METHOD FB_init : BOOL
VAR_INPUT
	bInitRetains : BOOL; // if TRUE, the retain variables are initialized (warm start / cold start)
	bInCopyCode : BOOL;  // if TRUE, the instance afterwards gets moved into the copy code (online change)
	InitialValue : ETcVnReduceType;
END_VAR
localData := InitialValue;
AddBaseDatatype(enumBaseDatatype);
ClearReference();

AddLocalEnumeration('TCVN_RT_REDUCE_SUM', ETcVnReduceType.TCVN_RT_REDUCE_SUM);
AddLocalEnumeration('TCVN_RT_REDUCE_AVG', ETcVnReduceType.TCVN_RT_REDUCE_AVG);
AddLocalEnumeration('TCVN_RT_REDUCE_MAX', ETcVnReduceType.TCVN_RT_REDUCE_MAX);
AddLocalEnumeration('TCVN_RT_REDUCE_MIN', ETcVnReduceType.TCVN_RT_REDUCE_MIN);
END_METHOD

METHOD PRIVATE AddLocalEnumeration
VAR_INPUT
	Enumeration : T_MAXSTRING;
	Value : ETcVnReduceType;
END_VAR
AddEnumeration(Enumeration, Value);
END_METHOD

METHOD IsEnumeratorValueEqual : BOOL
VAR_INPUT
	Enumerator : I_KeyValueForwardEnumerator;
END_VAR
VAR
	storedValue : ETcVnReduceType;
END_VAR
IF NOT Enumerator.TryGet(storedValue) THEN
	RETURN;
END_IF

IsEnumeratorValueEqual := storedValue = activeData;
END_METHOD

METHOD PUBLIC Clone : I_Datatype
VAR
    pClone : POINTER TO _ETcVnReduceType;
END_VAR
pClone := __NEW(_ETcVnReduceType(InitialValue := Value));
Clone := pClone^;
END_METHOD

PROPERTY PUBLIC Identifier : T_MAXSTRING
GET
Identifier := 'ETcVnReduceType';
END_GET
END_PROPERTY

METHOD PUBLIC MakeReferenceTo
VAR_INPUT
	ReferenceTarget : REFERENCE TO ETcVnReduceType;
END_VAR
activeData REF= ReferenceTarget;
SetBaseDatatypeReference();
END_METHOD

METHOD TryMakeReferenceTo : BOOL
VAR_INPUT
	Target : I_Datatype;
END_VAR
VAR
	pTargetData : POINTER TO ETcVnReduceType;
END_VAR
IF NOT IsEquivalentTo(Target) THEN
	RETURN;
END_IF

pTargetData := Target.Address;
activeData REF= pTargetData^;
SetBaseDatatypeReference();
TryMakeReferenceTo := TRUE;
END_METHOD

PROPERTY PUBLIC Value : ETcVnReduceType
GET
Value := activeData;
END_GET
SET
activeData := Value;
END_SET
END_PROPERTY

END_FUNCTION_BLOCK

// Datatypes/Enums/_ETcVnRotationAngle
{attribute 'linkalways'} 
{attribute 'no_explicit_call' := 'This FB is a CLASS and must be accessed using methods or properties'}
{attribute 'enable_dynamic_creation'}
FUNCTION_BLOCK _ETcVnRotationAngle EXTENDS EnumDatatypeBase
VAR
	localData : ETcVnRotationAngle;
	activeData : REFERENCE TO ETcVnRotationAngle;
	enumBaseDatatype : _DINT(localData);
END_VAR

METHOD PROTECTED SetBaseDatatypeReference
VAR_INPUT
END_VAR
enumBaseDatatype.MakeReferenceTo(activeData);
END_METHOD

PROPERTY PUBLIC Address : PVOID
GET
Address := ADR(activeData);
END_GET
END_PROPERTY

METHOD PUBLIC ClearReference
VAR_INPUT
END_VAR
activeData REF= localData;
SetBaseDatatypeReference();
END_METHOD

PROPERTY PUBLIC Size : UDINT
GET
Size := SIZEOF(activeData);
END_GET
END_PROPERTY

METHOD FB_init : BOOL
VAR_INPUT
	bInitRetains : BOOL; // if TRUE, the retain variables are initialized (warm start / cold start)
	bInCopyCode : BOOL;  // if TRUE, the instance afterwards gets moved into the copy code (online change)
	InitialValue : ETcVnRotationAngle;
END_VAR
localData := InitialValue;
AddBaseDatatype(enumBaseDatatype);
ClearReference();

AddLocalEnumeration('TCVN_RA_90_DEG', ETcVnRotationAngle.TCVN_RA_90_DEG);
AddLocalEnumeration('TCVN_RA_180_DEG', ETcVnRotationAngle.TCVN_RA_180_DEG);
AddLocalEnumeration('TCVN_RA_270_DEG', ETcVnRotationAngle.TCVN_RA_270_DEG);
END_METHOD

METHOD PRIVATE AddLocalEnumeration
VAR_INPUT
	Enumeration : T_MAXSTRING;
	Value : ETcVnRotationAngle;
END_VAR
AddEnumeration(Enumeration, Value);
END_METHOD

METHOD IsEnumeratorValueEqual : BOOL
VAR_INPUT
	Enumerator : I_KeyValueForwardEnumerator;
END_VAR
VAR
	storedValue : ETcVnRotationAngle;
END_VAR
IF NOT Enumerator.TryGet(storedValue) THEN
	RETURN;
END_IF

IsEnumeratorValueEqual := storedValue = activeData;
END_METHOD

METHOD PUBLIC Clone : I_Datatype
VAR
    pClone : POINTER TO _ETcVnRotationAngle;
END_VAR
pClone := __NEW(_ETcVnRotationAngle(InitialValue := Value));
Clone := pClone^;
END_METHOD

PROPERTY PUBLIC Identifier : T_MAXSTRING
GET
Identifier := 'ETcVnRotationAngle';
END_GET
END_PROPERTY

METHOD PUBLIC MakeReferenceTo
VAR_INPUT
	ReferenceTarget : REFERENCE TO ETcVnRotationAngle;
END_VAR
activeData REF= ReferenceTarget;
SetBaseDatatypeReference();
END_METHOD

METHOD TryMakeReferenceTo : BOOL
VAR_INPUT
	Target : I_Datatype;
END_VAR
VAR
	pTargetData : POINTER TO ETcVnRotationAngle;
END_VAR
IF NOT IsEquivalentTo(Target) THEN
	RETURN;
END_IF

pTargetData := Target.Address;
activeData REF= pTargetData^;
SetBaseDatatypeReference();
TryMakeReferenceTo := TRUE;
END_METHOD

PROPERTY PUBLIC Value : ETcVnRotationAngle
GET
Value := activeData;
END_GET
SET
activeData := Value;
END_SET
END_PROPERTY

END_FUNCTION_BLOCK

// Datatypes/Enums/_ETcVnRTrees
{attribute 'linkalways'} 
{attribute 'no_explicit_call' := 'This FB is a CLASS and must be accessed using methods or properties'}
{attribute 'enable_dynamic_creation'}
FUNCTION_BLOCK _ETcVnRTrees EXTENDS EnumDatatypeBase
VAR
	localData : ETcVnRTrees;
	activeData : REFERENCE TO ETcVnRTrees;
	enumBaseDatatype : _UDINT(localData);
END_VAR

METHOD PROTECTED SetBaseDatatypeReference
VAR_INPUT
END_VAR
enumBaseDatatype.MakeReferenceTo(activeData);
END_METHOD

PROPERTY PUBLIC Address : PVOID
GET
Address := ADR(activeData);
END_GET
END_PROPERTY

METHOD PUBLIC ClearReference
VAR_INPUT
END_VAR
activeData REF= localData;
SetBaseDatatypeReference();
END_METHOD

PROPERTY PUBLIC Size : UDINT
GET
Size := SIZEOF(activeData);
END_GET
END_PROPERTY

METHOD FB_init : BOOL
VAR_INPUT
	bInitRetains : BOOL; // if TRUE, the retain variables are initialized (warm start / cold start)
	bInCopyCode : BOOL;  // if TRUE, the instance afterwards gets moved into the copy code (online change)
	InitialValue : ETcVnRTrees;
END_VAR
localData := InitialValue;
AddBaseDatatype(enumBaseDatatype);
ClearReference();

AddLocalEnumeration('TCVN_RT_CLASSIFIER', ETcVnRTrees.TCVN_RT_CLASSIFIER);
AddLocalEnumeration('TCVN_RT_REGRESSOR', ETcVnRTrees.TCVN_RT_REGRESSOR);
END_METHOD

METHOD PRIVATE AddLocalEnumeration
VAR_INPUT
	Enumeration : T_MAXSTRING;
	Value : ETcVnRTrees;
END_VAR
AddEnumeration(Enumeration, Value);
END_METHOD

METHOD IsEnumeratorValueEqual : BOOL
VAR_INPUT
	Enumerator : I_KeyValueForwardEnumerator;
END_VAR
VAR
	storedValue : ETcVnRTrees;
END_VAR
IF NOT Enumerator.TryGet(storedValue) THEN
	RETURN;
END_IF

IsEnumeratorValueEqual := storedValue = activeData;
END_METHOD

METHOD PUBLIC Clone : I_Datatype
VAR
    pClone : POINTER TO _ETcVnRTrees;
END_VAR
pClone := __NEW(_ETcVnRTrees(InitialValue := Value));
Clone := pClone^;
END_METHOD

PROPERTY PUBLIC Identifier : T_MAXSTRING
GET
Identifier := 'ETcVnRTrees';
END_GET
END_PROPERTY

METHOD PUBLIC MakeReferenceTo
VAR_INPUT
	ReferenceTarget : REFERENCE TO ETcVnRTrees;
END_VAR
activeData REF= ReferenceTarget;
SetBaseDatatypeReference();
END_METHOD

METHOD TryMakeReferenceTo : BOOL
VAR_INPUT
	Target : I_Datatype;
END_VAR
VAR
	pTargetData : POINTER TO ETcVnRTrees;
END_VAR
IF NOT IsEquivalentTo(Target) THEN
	RETURN;
END_IF

pTargetData := Target.Address;
activeData REF= pTargetData^;
SetBaseDatatypeReference();
TryMakeReferenceTo := TRUE;
END_METHOD

PROPERTY PUBLIC Value : ETcVnRTrees
GET
Value := activeData;
END_GET
SET
activeData := Value;
END_SET
END_PROPERTY

END_FUNCTION_BLOCK

// Datatypes/Enums/_ETcVnSalientFeaturesMethod
{attribute 'linkalways'}
{attribute 'no_explicit_call' := 'This FB is a CLASS and must be accessed using methods or properties'}
{attribute 'enable_dynamic_creation'}
FUNCTION_BLOCK _ETcVnSalientFeaturesMethod EXTENDS EnumDatatypeBase
VAR
	localData : ETcVnSalientFeaturesMethod;
	activeData : REFERENCE TO ETcVnSalientFeaturesMethod;
	enumBaseDatatype : _UDINT(localData);
END_VAR

METHOD PROTECTED SetBaseDatatypeReference
VAR_INPUT
END_VAR
enumBaseDatatype.MakeReferenceTo(activeData);
END_METHOD

PROPERTY PUBLIC Address : PVOID
GET
Address := ADR(activeData);
END_GET
END_PROPERTY

METHOD PUBLIC ClearReference
VAR_INPUT
END_VAR
activeData REF= localData;
SetBaseDatatypeReference();
END_METHOD

PROPERTY PUBLIC Size : UDINT
GET
Size := SIZEOF(activeData);
END_GET
END_PROPERTY

METHOD FB_init : BOOL
VAR_INPUT
	bInitRetains : BOOL; // if TRUE, the retain variables are initialized (warm start / cold start)
	bInCopyCode : BOOL;  // if TRUE, the instance afterwards gets moved into the copy code (online change)
	InitialValue : ETcVnSalientFeaturesMethod;
END_VAR
localData := InitialValue;
AddBaseDatatype(enumBaseDatatype);
ClearReference();

AddLocalEnumeration('TCVN_SFM_WALSH_CODE', ETcVnSalientFeaturesMethod.TCVN_SFM_WALSH_CODE);
AddLocalEnumeration('TCVN_SFM_SOBEL', ETcVnSalientFeaturesMethod.TCVN_SFM_SOBEL);
END_METHOD

METHOD PRIVATE AddLocalEnumeration
VAR_INPUT
	Enumeration : T_MAXSTRING;
	Value : ETcVnSalientFeaturesMethod;
END_VAR
AddEnumeration(Enumeration, Value);
END_METHOD

METHOD IsEnumeratorValueEqual : BOOL
VAR_INPUT
	Enumerator : I_KeyValueForwardEnumerator;
END_VAR
VAR
	storedValue : ETcVnSalientFeaturesMethod;
END_VAR
IF NOT Enumerator.TryGet(storedValue) THEN
	RETURN;
END_IF

IsEnumeratorValueEqual := storedValue = activeData;
END_METHOD

METHOD PUBLIC Clone : I_Datatype
VAR
    pClone : POINTER TO _ETcVnSalientFeaturesMethod;
END_VAR
pClone := __NEW(_ETcVnSalientFeaturesMethod(InitialValue := Value));
IF pClone = 0 THEN
    RETURN;
END_IF
Clone := pClone^;
END_METHOD

PROPERTY PUBLIC Identifier : T_MAXSTRING
GET
Identifier := 'ETcVnSalientFeaturesMethod';
END_GET
END_PROPERTY

METHOD PUBLIC MakeReferenceTo
VAR_INPUT
	ReferenceTarget : REFERENCE TO ETcVnSalientFeaturesMethod;
END_VAR
activeData REF= ReferenceTarget;
SetBaseDatatypeReference();
END_METHOD

METHOD TryMakeReferenceTo : BOOL
VAR_INPUT
	Target : I_Datatype;
END_VAR
VAR
	pTargetData : POINTER TO ETcVnSalientFeaturesMethod;
END_VAR
IF NOT IsEquivalentTo(Target) THEN
	RETURN;
END_IF

pTargetData := Target.Address;
activeData REF= pTargetData^;
SetBaseDatatypeReference();
TryMakeReferenceTo := TRUE;
END_METHOD

PROPERTY PUBLIC Value : ETcVnSalientFeaturesMethod
GET
Value := activeData;
END_GET
SET
activeData := Value;
END_SET
END_PROPERTY

END_FUNCTION_BLOCK

// Datatypes/Enums/_ETcVnSignedNormalization
{attribute 'linkalways'} 
{attribute 'no_explicit_call' := 'This FB is a CLASS and must be accessed using methods or properties'}
{attribute 'enable_dynamic_creation'}
FUNCTION_BLOCK _ETcVnSignedNormalization EXTENDS EnumDatatypeBase
VAR
	localData : ETcVnSignedNormalization;
	activeData : REFERENCE TO ETcVnSignedNormalization;
	enumBaseDatatype : _INT(localData);
END_VAR

METHOD PROTECTED SetBaseDatatypeReference
VAR_INPUT
END_VAR
enumBaseDatatype.MakeReferenceTo(activeData);
END_METHOD

PROPERTY PUBLIC Address : PVOID
GET
Address := ADR(activeData);
END_GET
END_PROPERTY

METHOD PUBLIC ClearReference
VAR_INPUT
END_VAR
activeData REF= localData;
SetBaseDatatypeReference();
END_METHOD

PROPERTY PUBLIC Size : UDINT
GET
Size := SIZEOF(activeData);
END_GET
END_PROPERTY

METHOD FB_init : BOOL
VAR_INPUT
	bInitRetains : BOOL; // if TRUE, the retain variables are initialized (warm start / cold start)
	bInCopyCode : BOOL;  // if TRUE, the instance afterwards gets moved into the copy code (online change)
	InitialValue : ETcVnSignedNormalization;
END_VAR
localData := InitialValue;
AddBaseDatatype(enumBaseDatatype);
ClearReference();

AddLocalEnumeration('TCVN_SN_FIX_ZERO', ETcVnSignedNormalization.TCVN_SN_FIX_ZERO);
AddLocalEnumeration('TCVN_SN_FULL_SCALE', ETcVnSignedNormalization.TCVN_SN_FULL_SCALE);
END_METHOD

METHOD PRIVATE AddLocalEnumeration
VAR_INPUT
	Enumeration : T_MAXSTRING;
	Value : ETcVnSignedNormalization;
END_VAR
AddEnumeration(Enumeration, Value);
END_METHOD

METHOD IsEnumeratorValueEqual : BOOL
VAR_INPUT
	Enumerator : I_KeyValueForwardEnumerator;
END_VAR
VAR
	storedValue : ETcVnSignedNormalization;
END_VAR
IF NOT Enumerator.TryGet(storedValue) THEN
	RETURN;
END_IF

IsEnumeratorValueEqual := storedValue = activeData;
END_METHOD

METHOD PUBLIC Clone : I_Datatype
VAR
    pClone : POINTER TO _ETcVnSignedNormalization;
END_VAR
pClone := __NEW(_ETcVnSignedNormalization(InitialValue := Value));
Clone := pClone^;
END_METHOD

PROPERTY PUBLIC Identifier : T_MAXSTRING
GET
Identifier := 'ETcVnSignedNormalization';
END_GET
END_PROPERTY

METHOD PUBLIC MakeReferenceTo
VAR_INPUT
	ReferenceTarget : REFERENCE TO ETcVnSignedNormalization;
END_VAR
activeData REF= ReferenceTarget;
SetBaseDatatypeReference();
END_METHOD

METHOD TryMakeReferenceTo : BOOL
VAR_INPUT
	Target : I_Datatype;
END_VAR
VAR
	pTargetData : POINTER TO ETcVnSignedNormalization;
END_VAR
IF NOT IsEquivalentTo(Target) THEN
	RETURN;
END_IF

pTargetData := Target.Address;
activeData REF= pTargetData^;
SetBaseDatatypeReference();
TryMakeReferenceTo := TRUE;
END_METHOD

PROPERTY PUBLIC Value : ETcVnSignedNormalization
GET
Value := activeData;
END_GET
SET
activeData := Value;
END_SET
END_PROPERTY

END_FUNCTION_BLOCK

// Datatypes/Enums/_ETcVnSolvePnPMethod
{attribute 'linkalways'} 
{attribute 'no_explicit_call' := 'This FB is a CLASS and must be accessed using methods or properties'}
{attribute 'enable_dynamic_creation'}
FUNCTION_BLOCK _ETcVnSolvePnPMethod EXTENDS EnumDatatypeBase
VAR
	localData : ETcVnSolvePnPMethod;
	activeData : REFERENCE TO ETcVnSolvePnPMethod;
	enumBaseDatatype : _DINT(localData);
END_VAR

METHOD PROTECTED SetBaseDatatypeReference
VAR_INPUT
END_VAR
enumBaseDatatype.MakeReferenceTo(activeData);
END_METHOD

PROPERTY PUBLIC Address : PVOID
GET
Address := ADR(activeData);
END_GET
END_PROPERTY

METHOD PUBLIC ClearReference
VAR_INPUT
END_VAR
activeData REF= localData;
SetBaseDatatypeReference();
END_METHOD

PROPERTY PUBLIC Size : UDINT
GET
Size := SIZEOF(activeData);
END_GET
END_PROPERTY

METHOD FB_init : BOOL
VAR_INPUT
	bInitRetains : BOOL; // if TRUE, the retain variables are initialized (warm start / cold start)
	bInCopyCode : BOOL;  // if TRUE, the instance afterwards gets moved into the copy code (online change)
	InitialValue : ETcVnSolvePnPMethod;
END_VAR
localData := InitialValue;
AddBaseDatatype(enumBaseDatatype);
ClearReference();

AddLocalEnumeration('TCVN_SPM_ITERATIVE', ETcVnSolvePnPMethod.TCVN_SPM_ITERATIVE);
AddLocalEnumeration('TCVN_SPM_EPNP', ETcVnSolvePnPMethod.TCVN_SPM_EPNP);
AddLocalEnumeration('TCVN_SPM_P3P', ETcVnSolvePnPMethod.TCVN_SPM_P3P);
AddLocalEnumeration('TCVN_SPM_AP3P', ETcVnSolvePnPMethod.TCVN_SPM_AP3P);
AddLocalEnumeration('TCVN_SPM_IPPE', ETcVnSolvePnPMethod.TCVN_SPM_IPPE);
AddLocalEnumeration('TCVN_SPM_IPPE_SQUARE', ETcVnSolvePnPMethod.TCVN_SPM_IPPE_SQUARE);
AddLocalEnumeration('TCVN_SPM_SQPNP', ETcVnSolvePnPMethod.TCVN_SPM_SQPNP);
END_METHOD

METHOD PRIVATE AddLocalEnumeration
VAR_INPUT
	Enumeration : T_MAXSTRING;
	Value : ETcVnSolvePnPMethod;
END_VAR
AddEnumeration(Enumeration, Value);
END_METHOD

METHOD IsEnumeratorValueEqual : BOOL
VAR_INPUT
	Enumerator : I_KeyValueForwardEnumerator;
END_VAR
VAR
	storedValue : ETcVnSolvePnPMethod;
END_VAR
IF NOT Enumerator.TryGet(storedValue) THEN
	RETURN;
END_IF

IsEnumeratorValueEqual := storedValue = activeData;
END_METHOD

METHOD PUBLIC Clone : I_Datatype
VAR
    pClone : POINTER TO _ETcVnSolvePnPMethod;
END_VAR
pClone := __NEW(_ETcVnSolvePnPMethod(InitialValue := Value));
Clone := pClone^;
END_METHOD

PROPERTY PUBLIC Identifier : T_MAXSTRING
GET
Identifier := 'ETcVnSolvePnPMethod';
END_GET
END_PROPERTY

METHOD PUBLIC MakeReferenceTo
VAR_INPUT
	ReferenceTarget : REFERENCE TO ETcVnSolvePnPMethod;
END_VAR
activeData REF= ReferenceTarget;
SetBaseDatatypeReference();
END_METHOD

METHOD TryMakeReferenceTo : BOOL
VAR_INPUT
	Target : I_Datatype;
END_VAR
VAR
	pTargetData : POINTER TO ETcVnSolvePnPMethod;
END_VAR
IF NOT IsEquivalentTo(Target) THEN
	RETURN;
END_IF

pTargetData := Target.Address;
activeData REF= pTargetData^;
SetBaseDatatypeReference();
TryMakeReferenceTo := TRUE;
END_METHOD

PROPERTY PUBLIC Value : ETcVnSolvePnPMethod
GET
Value := activeData;
END_GET
SET
activeData := Value;
END_SET
END_PROPERTY

END_FUNCTION_BLOCK

// Datatypes/Enums/_ETcVnSta
{attribute 'linkalways'} 
{attribute 'no_explicit_call' := 'This FB is a CLASS and must be accessed using methods or properties'}
{attribute 'enable_dynamic_creation'}
FUNCTION_BLOCK _ETcVnSta EXTENDS EnumDatatypeBase
VAR
	localData : ETcVnSta;
	activeData : REFERENCE TO ETcVnSta;
	enumBaseDatatype : _UDINT(localData);
END_VAR

METHOD PROTECTED SetBaseDatatypeReference
VAR_INPUT
END_VAR
enumBaseDatatype.MakeReferenceTo(activeData);
END_METHOD

PROPERTY PUBLIC Address : PVOID
GET
Address := ADR(activeData);
END_GET
END_PROPERTY

METHOD PUBLIC ClearReference
VAR_INPUT
END_VAR
activeData REF= localData;
SetBaseDatatypeReference();
END_METHOD

PROPERTY PUBLIC Size : UDINT
GET
Size := SIZEOF(activeData);
END_GET
END_PROPERTY

METHOD FB_init : BOOL
VAR_INPUT
	bInitRetains : BOOL; // if TRUE, the retain variables are initialized (warm start / cold start)
	bInCopyCode : BOOL;  // if TRUE, the instance afterwards gets moved into the copy code (online change)
	InitialValue : ETcVnSta;
END_VAR
localData := InitialValue;
AddBaseDatatype(enumBaseDatatype);
ClearReference();

AddLocalEnumeration('TCVN_STA_CLASSIFIER', ETcVnSta.TCVN_STA_CLASSIFIER);
AddLocalEnumeration('TCVN_STA_NOVELTY_DETECTOR', ETcVnSta.TCVN_STA_NOVELTY_DETECTOR);
AddLocalEnumeration('TCVN_STA_REGRESSOR', ETcVnSta.TCVN_STA_REGRESSOR);
AddLocalEnumeration('TCVN_STA_CLUSTERER', ETcVnSta.TCVN_STA_CLUSTERER);
END_METHOD

METHOD PRIVATE AddLocalEnumeration
VAR_INPUT
	Enumeration : T_MAXSTRING;
	Value : ETcVnSta;
END_VAR
AddEnumeration(Enumeration, Value);
END_METHOD

METHOD IsEnumeratorValueEqual : BOOL
VAR_INPUT
	Enumerator : I_KeyValueForwardEnumerator;
END_VAR
VAR
	storedValue : ETcVnSta;
END_VAR
IF NOT Enumerator.TryGet(storedValue) THEN
	RETURN;
END_IF

IsEnumeratorValueEqual := storedValue = activeData;
END_METHOD

METHOD PUBLIC Clone : I_Datatype
VAR
    pClone : POINTER TO _ETcVnSta;
END_VAR
pClone := __NEW(_ETcVnSta(InitialValue := Value));
Clone := pClone^;
END_METHOD

PROPERTY PUBLIC Identifier : T_MAXSTRING
GET
Identifier := 'ETcVnSta';
END_GET
END_PROPERTY

METHOD PUBLIC MakeReferenceTo
VAR_INPUT
	ReferenceTarget : REFERENCE TO ETcVnSta;
END_VAR
activeData REF= ReferenceTarget;
SetBaseDatatypeReference();
END_METHOD

METHOD TryMakeReferenceTo : BOOL
VAR_INPUT
	Target : I_Datatype;
END_VAR
VAR
	pTargetData : POINTER TO ETcVnSta;
END_VAR
IF NOT IsEquivalentTo(Target) THEN
	RETURN;
END_IF

pTargetData := Target.Address;
activeData REF= pTargetData^;
SetBaseDatatypeReference();
TryMakeReferenceTo := TRUE;
END_METHOD

PROPERTY PUBLIC Value : ETcVnSta
GET
Value := activeData;
END_GET
SET
activeData := Value;
END_SET
END_PROPERTY

END_FUNCTION_BLOCK

// Datatypes/Enums/_ETcVnStructuringElementShape
{attribute 'linkalways'} 
{attribute 'no_explicit_call' := 'This FB is a CLASS and must be accessed using methods or properties'}
{attribute 'enable_dynamic_creation'}
FUNCTION_BLOCK _ETcVnStructuringElementShape EXTENDS EnumDatatypeBase
VAR
	localData : ETcVnStructuringElementShape;
	activeData : REFERENCE TO ETcVnStructuringElementShape;
	enumBaseDatatype : _DINT(localData);
END_VAR

METHOD PROTECTED SetBaseDatatypeReference
VAR_INPUT
END_VAR
enumBaseDatatype.MakeReferenceTo(activeData);
END_METHOD

PROPERTY PUBLIC Address : PVOID
GET
Address := ADR(activeData);
END_GET
END_PROPERTY

METHOD PUBLIC ClearReference
VAR_INPUT
END_VAR
activeData REF= localData;
SetBaseDatatypeReference();
END_METHOD

PROPERTY PUBLIC Size : UDINT
GET
Size := SIZEOF(activeData);
END_GET
END_PROPERTY

METHOD FB_init : BOOL
VAR_INPUT
	bInitRetains : BOOL; // if TRUE, the retain variables are initialized (warm start / cold start)
	bInCopyCode : BOOL;  // if TRUE, the instance afterwards gets moved into the copy code (online change)
	InitialValue : ETcVnStructuringElementShape;
END_VAR
localData := InitialValue;
AddBaseDatatype(enumBaseDatatype);
ClearReference();

AddLocalEnumeration('TCVN_SES_RECTANGLE', ETcVnStructuringElementShape.TCVN_SES_RECTANGLE);
AddLocalEnumeration('TCVN_SES_CROSS', ETcVnStructuringElementShape.TCVN_SES_CROSS);
AddLocalEnumeration('TCVN_SES_ELLIPSE', ETcVnStructuringElementShape.TCVN_SES_ELLIPSE);
END_METHOD

METHOD PRIVATE AddLocalEnumeration
VAR_INPUT
	Enumeration : T_MAXSTRING;
	Value : ETcVnStructuringElementShape;
END_VAR
AddEnumeration(Enumeration, Value);
END_METHOD

METHOD IsEnumeratorValueEqual : BOOL
VAR_INPUT
	Enumerator : I_KeyValueForwardEnumerator;
END_VAR
VAR
	storedValue : ETcVnStructuringElementShape;
END_VAR
IF NOT Enumerator.TryGet(storedValue) THEN
	RETURN;
END_IF

IsEnumeratorValueEqual := storedValue = activeData;
END_METHOD

METHOD PUBLIC Clone : I_Datatype
VAR
    pClone : POINTER TO _ETcVnStructuringElementShape;
END_VAR
pClone := __NEW(_ETcVnStructuringElementShape(InitialValue := Value));
Clone := pClone^;
END_METHOD

PROPERTY PUBLIC Identifier : T_MAXSTRING
GET
Identifier := 'ETcVnStructuringElementShape';
END_GET
END_PROPERTY

METHOD PUBLIC MakeReferenceTo
VAR_INPUT
	ReferenceTarget : REFERENCE TO ETcVnStructuringElementShape;
END_VAR
activeData REF= ReferenceTarget;
SetBaseDatatypeReference();
END_METHOD

METHOD TryMakeReferenceTo : BOOL
VAR_INPUT
	Target : I_Datatype;
END_VAR
VAR
	pTargetData : POINTER TO ETcVnStructuringElementShape;
END_VAR
IF NOT IsEquivalentTo(Target) THEN
	RETURN;
END_IF

pTargetData := Target.Address;
activeData REF= pTargetData^;
SetBaseDatatypeReference();
TryMakeReferenceTo := TRUE;
END_METHOD

PROPERTY PUBLIC Value : ETcVnStructuringElementShape
GET
Value := activeData;
END_GET
SET
activeData := Value;
END_SET
END_PROPERTY

END_FUNCTION_BLOCK

// Datatypes/Enums/_ETcVnSvm
{attribute 'linkalways'} 
{attribute 'no_explicit_call' := 'This FB is a CLASS and must be accessed using methods or properties'}
{attribute 'enable_dynamic_creation'}
FUNCTION_BLOCK _ETcVnSvm EXTENDS EnumDatatypeBase
VAR
	localData : ETcVnSvm;
	activeData : REFERENCE TO ETcVnSvm;
	enumBaseDatatype : _UDINT(localData);
END_VAR

METHOD PROTECTED SetBaseDatatypeReference
VAR_INPUT
END_VAR
enumBaseDatatype.MakeReferenceTo(activeData);
END_METHOD

PROPERTY PUBLIC Address : PVOID
GET
Address := ADR(activeData);
END_GET
END_PROPERTY

METHOD PUBLIC ClearReference
VAR_INPUT
END_VAR
activeData REF= localData;
SetBaseDatatypeReference();
END_METHOD

PROPERTY PUBLIC Size : UDINT
GET
Size := SIZEOF(activeData);
END_GET
END_PROPERTY

METHOD FB_init : BOOL
VAR_INPUT
	bInitRetains : BOOL; // if TRUE, the retain variables are initialized (warm start / cold start)
	bInCopyCode : BOOL;  // if TRUE, the instance afterwards gets moved into the copy code (online change)
	InitialValue : ETcVnSvm;
END_VAR
localData := InitialValue;
AddBaseDatatype(enumBaseDatatype);
ClearReference();

AddLocalEnumeration('TCVN_SVM_C_CLASSIFIER', ETcVnSvm.TCVN_SVM_C_CLASSIFIER);
AddLocalEnumeration('TCVN_SVM_NU_CLASSIFIER', ETcVnSvm.TCVN_SVM_NU_CLASSIFIER);
AddLocalEnumeration('TCVN_SVM_NOVELTY_DETECTOR', ETcVnSvm.TCVN_SVM_NOVELTY_DETECTOR);
AddLocalEnumeration('TCVN_SVM_EPS_REGRESSOR', ETcVnSvm.TCVN_SVM_EPS_REGRESSOR);
AddLocalEnumeration('TCVN_SVM_NU_REGRESSOR', ETcVnSvm.TCVN_SVM_NU_REGRESSOR);
END_METHOD

METHOD PRIVATE AddLocalEnumeration
VAR_INPUT
	Enumeration : T_MAXSTRING;
	Value : ETcVnSvm;
END_VAR
AddEnumeration(Enumeration, Value);
END_METHOD

METHOD IsEnumeratorValueEqual : BOOL
VAR_INPUT
	Enumerator : I_KeyValueForwardEnumerator;
END_VAR
VAR
	storedValue : ETcVnSvm;
END_VAR
IF NOT Enumerator.TryGet(storedValue) THEN
	RETURN;
END_IF

IsEnumeratorValueEqual := storedValue = activeData;
END_METHOD

METHOD PUBLIC Clone : I_Datatype
VAR
    pClone : POINTER TO _ETcVnSvm;
END_VAR
pClone := __NEW(_ETcVnSvm(InitialValue := Value));
Clone := pClone^;
END_METHOD

PROPERTY PUBLIC Identifier : T_MAXSTRING
GET
Identifier := 'ETcVnSvm';
END_GET
END_PROPERTY

METHOD PUBLIC MakeReferenceTo
VAR_INPUT
	ReferenceTarget : REFERENCE TO ETcVnSvm;
END_VAR
activeData REF= ReferenceTarget;
SetBaseDatatypeReference();
END_METHOD

METHOD TryMakeReferenceTo : BOOL
VAR_INPUT
	Target : I_Datatype;
END_VAR
VAR
	pTargetData : POINTER TO ETcVnSvm;
END_VAR
IF NOT IsEquivalentTo(Target) THEN
	RETURN;
END_IF

pTargetData := Target.Address;
activeData REF= pTargetData^;
SetBaseDatatypeReference();
TryMakeReferenceTo := TRUE;
END_METHOD

PROPERTY PUBLIC Value : ETcVnSvm
GET
Value := activeData;
END_GET
SET
activeData := Value;
END_SET
END_PROPERTY

END_FUNCTION_BLOCK

// Datatypes/Enums/_ETcVnSvmKernelType
{attribute 'linkalways'} 
{attribute 'no_explicit_call' := 'This FB is a CLASS and must be accessed using methods or properties'}
{attribute 'enable_dynamic_creation'}
FUNCTION_BLOCK _ETcVnSvmKernelType EXTENDS EnumDatatypeBase
VAR
	localData : ETcVnSvmKernelType;
	activeData : REFERENCE TO ETcVnSvmKernelType;
	enumBaseDatatype : _DINT(localData);
END_VAR

METHOD PROTECTED SetBaseDatatypeReference
VAR_INPUT
END_VAR
enumBaseDatatype.MakeReferenceTo(activeData);
END_METHOD

PROPERTY PUBLIC Address : PVOID
GET
Address := ADR(activeData);
END_GET
END_PROPERTY

METHOD PUBLIC ClearReference
VAR_INPUT
END_VAR
activeData REF= localData;
SetBaseDatatypeReference();
END_METHOD

PROPERTY PUBLIC Size : UDINT
GET
Size := SIZEOF(activeData);
END_GET
END_PROPERTY

METHOD FB_init : BOOL
VAR_INPUT
	bInitRetains : BOOL; // if TRUE, the retain variables are initialized (warm start / cold start)
	bInCopyCode : BOOL;  // if TRUE, the instance afterwards gets moved into the copy code (online change)
	InitialValue : ETcVnSvmKernelType;
END_VAR
localData := InitialValue;
AddBaseDatatype(enumBaseDatatype);
ClearReference();

AddLocalEnumeration('TCVN_SKT_LINEAR', ETcVnSvmKernelType.TCVN_SKT_LINEAR);
AddLocalEnumeration('TCVN_SKT_POLY', ETcVnSvmKernelType.TCVN_SKT_POLY);
AddLocalEnumeration('TCVN_SKT_RBF', ETcVnSvmKernelType.TCVN_SKT_RBF);
AddLocalEnumeration('TCVN_SKT_SIGMOID', ETcVnSvmKernelType.TCVN_SKT_SIGMOID);
AddLocalEnumeration('TCVN_SKT_CHI2', ETcVnSvmKernelType.TCVN_SKT_CHI2);
AddLocalEnumeration('TCVN_SKT_INTER', ETcVnSvmKernelType.TCVN_SKT_INTER);
END_METHOD

METHOD PRIVATE AddLocalEnumeration
VAR_INPUT
	Enumeration : T_MAXSTRING;
	Value : ETcVnSvmKernelType;
END_VAR
AddEnumeration(Enumeration, Value);
END_METHOD

METHOD IsEnumeratorValueEqual : BOOL
VAR_INPUT
	Enumerator : I_KeyValueForwardEnumerator;
END_VAR
VAR
	storedValue : ETcVnSvmKernelType;
END_VAR
IF NOT Enumerator.TryGet(storedValue) THEN
	RETURN;
END_IF

IsEnumeratorValueEqual := storedValue = activeData;
END_METHOD

METHOD PUBLIC Clone : I_Datatype
VAR
    pClone : POINTER TO _ETcVnSvmKernelType;
END_VAR
pClone := __NEW(_ETcVnSvmKernelType(InitialValue := Value));
Clone := pClone^;
END_METHOD

PROPERTY PUBLIC Identifier : T_MAXSTRING
GET
Identifier := 'ETcVnSvmKernelType';
END_GET
END_PROPERTY

METHOD PUBLIC MakeReferenceTo
VAR_INPUT
	ReferenceTarget : REFERENCE TO ETcVnSvmKernelType;
END_VAR
activeData REF= ReferenceTarget;
SetBaseDatatypeReference();
END_METHOD

METHOD TryMakeReferenceTo : BOOL
VAR_INPUT
	Target : I_Datatype;
END_VAR
VAR
	pTargetData : POINTER TO ETcVnSvmKernelType;
END_VAR
IF NOT IsEquivalentTo(Target) THEN
	RETURN;
END_IF

pTargetData := Target.Address;
activeData REF= pTargetData^;
SetBaseDatatypeReference();
TryMakeReferenceTo := TRUE;
END_METHOD

PROPERTY PUBLIC Value : ETcVnSvmKernelType
GET
Value := activeData;
END_GET
SET
activeData := Value;
END_SET
END_PROPERTY

END_FUNCTION_BLOCK

// Datatypes/Enums/_ETcVnSvmSgdClassifierMarginType
{attribute 'linkalways'} 
{attribute 'no_explicit_call' := 'This FB is a CLASS and must be accessed using methods or properties'}
{attribute 'enable_dynamic_creation'}
FUNCTION_BLOCK _ETcVnSvmSgdClassifierMarginType EXTENDS EnumDatatypeBase
VAR
	localData : ETcVnSvmSgdClassifierMarginType;
	activeData : REFERENCE TO ETcVnSvmSgdClassifierMarginType;
	enumBaseDatatype : _DINT(localData);
END_VAR

METHOD PROTECTED SetBaseDatatypeReference
VAR_INPUT
END_VAR
enumBaseDatatype.MakeReferenceTo(activeData);
END_METHOD

PROPERTY PUBLIC Address : PVOID
GET
Address := ADR(activeData);
END_GET
END_PROPERTY

METHOD PUBLIC ClearReference
VAR_INPUT
END_VAR
activeData REF= localData;
SetBaseDatatypeReference();
END_METHOD

PROPERTY PUBLIC Size : UDINT
GET
Size := SIZEOF(activeData);
END_GET
END_PROPERTY

METHOD FB_init : BOOL
VAR_INPUT
	bInitRetains : BOOL; // if TRUE, the retain variables are initialized (warm start / cold start)
	bInCopyCode : BOOL;  // if TRUE, the instance afterwards gets moved into the copy code (online change)
	InitialValue : ETcVnSvmSgdClassifierMarginType;
END_VAR
localData := InitialValue;
AddBaseDatatype(enumBaseDatatype);
ClearReference();

AddLocalEnumeration('TCVN_SSCMT_SOFT_MARGIN', ETcVnSvmSgdClassifierMarginType.TCVN_SSCMT_SOFT_MARGIN);
AddLocalEnumeration('TCVN_SSCMT_HARD_MARGIN', ETcVnSvmSgdClassifierMarginType.TCVN_SSCMT_HARD_MARGIN);
END_METHOD

METHOD PRIVATE AddLocalEnumeration
VAR_INPUT
	Enumeration : T_MAXSTRING;
	Value : ETcVnSvmSgdClassifierMarginType;
END_VAR
AddEnumeration(Enumeration, Value);
END_METHOD

METHOD IsEnumeratorValueEqual : BOOL
VAR_INPUT
	Enumerator : I_KeyValueForwardEnumerator;
END_VAR
VAR
	storedValue : ETcVnSvmSgdClassifierMarginType;
END_VAR
IF NOT Enumerator.TryGet(storedValue) THEN
	RETURN;
END_IF

IsEnumeratorValueEqual := storedValue = activeData;
END_METHOD

METHOD PUBLIC Clone : I_Datatype
VAR
    pClone : POINTER TO _ETcVnSvmSgdClassifierMarginType;
END_VAR
pClone := __NEW(_ETcVnSvmSgdClassifierMarginType(InitialValue := Value));
Clone := pClone^;
END_METHOD

PROPERTY PUBLIC Identifier : T_MAXSTRING
GET
Identifier := 'ETcVnSvmSgdClassifierMarginType';
END_GET
END_PROPERTY

METHOD PUBLIC MakeReferenceTo
VAR_INPUT
	ReferenceTarget : REFERENCE TO ETcVnSvmSgdClassifierMarginType;
END_VAR
activeData REF= ReferenceTarget;
SetBaseDatatypeReference();
END_METHOD

METHOD TryMakeReferenceTo : BOOL
VAR_INPUT
	Target : I_Datatype;
END_VAR
VAR
	pTargetData : POINTER TO ETcVnSvmSgdClassifierMarginType;
END_VAR
IF NOT IsEquivalentTo(Target) THEN
	RETURN;
END_IF

pTargetData := Target.Address;
activeData REF= pTargetData^;
SetBaseDatatypeReference();
TryMakeReferenceTo := TRUE;
END_METHOD

PROPERTY PUBLIC Value : ETcVnSvmSgdClassifierMarginType
GET
Value := activeData;
END_GET
SET
activeData := Value;
END_SET
END_PROPERTY

END_FUNCTION_BLOCK

// Datatypes/Enums/_ETcVnSvmSgdClassifierType
{attribute 'linkalways'} 
{attribute 'no_explicit_call' := 'This FB is a CLASS and must be accessed using methods or properties'}
{attribute 'enable_dynamic_creation'}
FUNCTION_BLOCK _ETcVnSvmSgdClassifierType EXTENDS EnumDatatypeBase
VAR
	localData : ETcVnSvmSgdClassifierType;
	activeData : REFERENCE TO ETcVnSvmSgdClassifierType;
	enumBaseDatatype : _DINT(localData);
END_VAR

METHOD PROTECTED SetBaseDatatypeReference
VAR_INPUT
END_VAR
enumBaseDatatype.MakeReferenceTo(activeData);
END_METHOD

PROPERTY PUBLIC Address : PVOID
GET
Address := ADR(activeData);
END_GET
END_PROPERTY

METHOD PUBLIC ClearReference
VAR_INPUT
END_VAR
activeData REF= localData;
SetBaseDatatypeReference();
END_METHOD

PROPERTY PUBLIC Size : UDINT
GET
Size := SIZEOF(activeData);
END_GET
END_PROPERTY

METHOD FB_init : BOOL
VAR_INPUT
	bInitRetains : BOOL; // if TRUE, the retain variables are initialized (warm start / cold start)
	bInCopyCode : BOOL;  // if TRUE, the instance afterwards gets moved into the copy code (online change)
	InitialValue : ETcVnSvmSgdClassifierType;
END_VAR
localData := InitialValue;
AddBaseDatatype(enumBaseDatatype);
ClearReference();

AddLocalEnumeration('TCVN_SSCT_SGD', ETcVnSvmSgdClassifierType.TCVN_SSCT_SGD);
AddLocalEnumeration('TCVN_SSCT_ASGD', ETcVnSvmSgdClassifierType.TCVN_SSCT_ASGD);
END_METHOD

METHOD PRIVATE AddLocalEnumeration
VAR_INPUT
	Enumeration : T_MAXSTRING;
	Value : ETcVnSvmSgdClassifierType;
END_VAR
AddEnumeration(Enumeration, Value);
END_METHOD

METHOD IsEnumeratorValueEqual : BOOL
VAR_INPUT
	Enumerator : I_KeyValueForwardEnumerator;
END_VAR
VAR
	storedValue : ETcVnSvmSgdClassifierType;
END_VAR
IF NOT Enumerator.TryGet(storedValue) THEN
	RETURN;
END_IF

IsEnumeratorValueEqual := storedValue = activeData;
END_METHOD

METHOD PUBLIC Clone : I_Datatype
VAR
    pClone : POINTER TO _ETcVnSvmSgdClassifierType;
END_VAR
pClone := __NEW(_ETcVnSvmSgdClassifierType(InitialValue := Value));
Clone := pClone^;
END_METHOD

PROPERTY PUBLIC Identifier : T_MAXSTRING
GET
Identifier := 'ETcVnSvmSgdClassifierType';
END_GET
END_PROPERTY

METHOD PUBLIC MakeReferenceTo
VAR_INPUT
	ReferenceTarget : REFERENCE TO ETcVnSvmSgdClassifierType;
END_VAR
activeData REF= ReferenceTarget;
SetBaseDatatypeReference();
END_METHOD

METHOD TryMakeReferenceTo : BOOL
VAR_INPUT
	Target : I_Datatype;
END_VAR
VAR
	pTargetData : POINTER TO ETcVnSvmSgdClassifierType;
END_VAR
IF NOT IsEquivalentTo(Target) THEN
	RETURN;
END_IF

pTargetData := Target.Address;
activeData REF= pTargetData^;
SetBaseDatatypeReference();
TryMakeReferenceTo := TRUE;
END_METHOD

PROPERTY PUBLIC Value : ETcVnSvmSgdClassifierType
GET
Value := activeData;
END_GET
SET
activeData := Value;
END_SET
END_PROPERTY

END_FUNCTION_BLOCK

// Datatypes/Enums/_ETcVnTemplateMatchMethod
{attribute 'linkalways'} 
{attribute 'no_explicit_call' := 'This FB is a CLASS and must be accessed using methods or properties'}
{attribute 'enable_dynamic_creation'}
FUNCTION_BLOCK _ETcVnTemplateMatchMethod EXTENDS EnumDatatypeBase
VAR
	localData : ETcVnTemplateMatchMethod;
	activeData : REFERENCE TO ETcVnTemplateMatchMethod;
	enumBaseDatatype : _DINT(localData);
END_VAR

METHOD PROTECTED SetBaseDatatypeReference
VAR_INPUT
END_VAR
enumBaseDatatype.MakeReferenceTo(activeData);
END_METHOD

PROPERTY PUBLIC Address : PVOID
GET
Address := ADR(activeData);
END_GET
END_PROPERTY

METHOD PUBLIC ClearReference
VAR_INPUT
END_VAR
activeData REF= localData;
SetBaseDatatypeReference();
END_METHOD

PROPERTY PUBLIC Size : UDINT
GET
Size := SIZEOF(activeData);
END_GET
END_PROPERTY

METHOD FB_init : BOOL
VAR_INPUT
	bInitRetains : BOOL; // if TRUE, the retain variables are initialized (warm start / cold start)
	bInCopyCode : BOOL;  // if TRUE, the instance afterwards gets moved into the copy code (online change)
	InitialValue : ETcVnTemplateMatchMethod;
END_VAR
localData := InitialValue;
AddBaseDatatype(enumBaseDatatype);
ClearReference();

AddLocalEnumeration('TCVN_TMM_SQDIFF', ETcVnTemplateMatchMethod.TCVN_TMM_SQDIFF);
AddLocalEnumeration('TCVN_TMM_SQDIFF_NORMED', ETcVnTemplateMatchMethod.TCVN_TMM_SQDIFF_NORMED);
AddLocalEnumeration('TCVN_TMM_CCORR', ETcVnTemplateMatchMethod.TCVN_TMM_CCORR);
AddLocalEnumeration('TCVN_TMM_CCORR_NORMED', ETcVnTemplateMatchMethod.TCVN_TMM_CCORR_NORMED);
AddLocalEnumeration('TCVN_TMM_CCOEFF', ETcVnTemplateMatchMethod.TCVN_TMM_CCOEFF);
AddLocalEnumeration('TCVN_TMM_CCOEFF_NORMED', ETcVnTemplateMatchMethod.TCVN_TMM_CCOEFF_NORMED);
END_METHOD

METHOD PRIVATE AddLocalEnumeration
VAR_INPUT
	Enumeration : T_MAXSTRING;
	Value : ETcVnTemplateMatchMethod;
END_VAR
AddEnumeration(Enumeration, Value);
END_METHOD

METHOD IsEnumeratorValueEqual : BOOL
VAR_INPUT
	Enumerator : I_KeyValueForwardEnumerator;
END_VAR
VAR
	storedValue : ETcVnTemplateMatchMethod;
END_VAR
IF NOT Enumerator.TryGet(storedValue) THEN
	RETURN;
END_IF

IsEnumeratorValueEqual := storedValue = activeData;
END_METHOD

METHOD PUBLIC Clone : I_Datatype
VAR
    pClone : POINTER TO _ETcVnTemplateMatchMethod;
END_VAR
pClone := __NEW(_ETcVnTemplateMatchMethod(InitialValue := Value));
Clone := pClone^;
END_METHOD

PROPERTY PUBLIC Identifier : T_MAXSTRING
GET
Identifier := 'ETcVnTemplateMatchMethod';
END_GET
END_PROPERTY

METHOD PUBLIC MakeReferenceTo
VAR_INPUT
	ReferenceTarget : REFERENCE TO ETcVnTemplateMatchMethod;
END_VAR
activeData REF= ReferenceTarget;
SetBaseDatatypeReference();
END_METHOD

METHOD TryMakeReferenceTo : BOOL
VAR_INPUT
	Target : I_Datatype;
END_VAR
VAR
	pTargetData : POINTER TO ETcVnTemplateMatchMethod;
END_VAR
IF NOT IsEquivalentTo(Target) THEN
	RETURN;
END_IF

pTargetData := Target.Address;
activeData REF= pTargetData^;
SetBaseDatatypeReference();
TryMakeReferenceTo := TRUE;
END_METHOD

PROPERTY PUBLIC Value : ETcVnTemplateMatchMethod
GET
Value := activeData;
END_GET
SET
activeData := Value;
END_SET
END_PROPERTY

END_FUNCTION_BLOCK

// Datatypes/Enums/_ETcVnThresholdType
{attribute 'linkalways'} 
{attribute 'no_explicit_call' := 'This FB is a CLASS and must be accessed using methods or properties'}
{attribute 'enable_dynamic_creation'}
FUNCTION_BLOCK _ETcVnThresholdType EXTENDS EnumDatatypeBase
VAR
	localData : ETcVnThresholdType;
	activeData : REFERENCE TO ETcVnThresholdType;
	enumBaseDatatype : _DINT(localData);
END_VAR

METHOD PROTECTED SetBaseDatatypeReference
VAR_INPUT
END_VAR
enumBaseDatatype.MakeReferenceTo(activeData);
END_METHOD

PROPERTY PUBLIC Address : PVOID
GET
Address := ADR(activeData);
END_GET
END_PROPERTY

METHOD PUBLIC ClearReference
VAR_INPUT
END_VAR
activeData REF= localData;
SetBaseDatatypeReference();
END_METHOD

PROPERTY PUBLIC Size : UDINT
GET
Size := SIZEOF(activeData);
END_GET
END_PROPERTY

METHOD FB_init : BOOL
VAR_INPUT
	bInitRetains : BOOL; // if TRUE, the retain variables are initialized (warm start / cold start)
	bInCopyCode : BOOL;  // if TRUE, the instance afterwards gets moved into the copy code (online change)
	InitialValue : ETcVnThresholdType;
END_VAR
localData := InitialValue;
AddBaseDatatype(enumBaseDatatype);
ClearReference();

AddLocalEnumeration('TCVN_TT_BINARY', ETcVnThresholdType.TCVN_TT_BINARY);
AddLocalEnumeration('TCVN_TT_BINARY_INV', ETcVnThresholdType.TCVN_TT_BINARY_INV);
AddLocalEnumeration('TCVN_TT_TRUNC', ETcVnThresholdType.TCVN_TT_TRUNC);
AddLocalEnumeration('TCVN_TT_TOZERO', ETcVnThresholdType.TCVN_TT_TOZERO);
AddLocalEnumeration('TCVN_TT_TOZERO_INV', ETcVnThresholdType.TCVN_TT_TOZERO_INV);
AddLocalEnumeration('TCVN_TT_OTSU_BINARY', ETcVnThresholdType.TCVN_TT_OTSU_BINARY);
AddLocalEnumeration('TCVN_TT_OTSU_BINARY_INV', ETcVnThresholdType.TCVN_TT_OTSU_BINARY_INV);
AddLocalEnumeration('TCVN_TT_OTSU_TRUNC', ETcVnThresholdType.TCVN_TT_OTSU_TRUNC);
AddLocalEnumeration('TCVN_TT_OTSU_TOZERO', ETcVnThresholdType.TCVN_TT_OTSU_TOZERO);
AddLocalEnumeration('TCVN_TT_OTSU_TOZERO_INV', ETcVnThresholdType.TCVN_TT_OTSU_TOZERO_INV);
AddLocalEnumeration('TCVN_TT_TRIANGLE_BINARY', ETcVnThresholdType.TCVN_TT_TRIANGLE_BINARY);
AddLocalEnumeration('TCVN_TT_TRIANGLE_BINARY_INV', ETcVnThresholdType.TCVN_TT_TRIANGLE_BINARY_INV);
AddLocalEnumeration('TCVN_TT_TRIANGLE_TRUNC', ETcVnThresholdType.TCVN_TT_TRIANGLE_TRUNC);
AddLocalEnumeration('TCVN_TT_TRIANGLE_TOZERO', ETcVnThresholdType.TCVN_TT_TRIANGLE_TOZERO);
AddLocalEnumeration('TCVN_TT_TRIANGLE_TOZERO_INV', ETcVnThresholdType.TCVN_TT_TRIANGLE_TOZERO_INV);
END_METHOD

METHOD PRIVATE AddLocalEnumeration
VAR_INPUT
	Enumeration : T_MAXSTRING;
	Value : ETcVnThresholdType;
END_VAR
AddEnumeration(Enumeration, Value);
END_METHOD

METHOD IsEnumeratorValueEqual : BOOL
VAR_INPUT
	Enumerator : I_KeyValueForwardEnumerator;
END_VAR
VAR
	storedValue : ETcVnThresholdType;
END_VAR
IF NOT Enumerator.TryGet(storedValue) THEN
	RETURN;
END_IF

IsEnumeratorValueEqual := storedValue = activeData;
END_METHOD

METHOD PUBLIC Clone : I_Datatype
VAR
    pClone : POINTER TO _ETcVnThresholdType;
END_VAR
pClone := __NEW(_ETcVnThresholdType(InitialValue := Value));
Clone := pClone^;
END_METHOD

PROPERTY PUBLIC Identifier : T_MAXSTRING
GET
Identifier := 'ETcVnThresholdType';
END_GET
END_PROPERTY

METHOD PUBLIC MakeReferenceTo
VAR_INPUT
	ReferenceTarget : REFERENCE TO ETcVnThresholdType;
END_VAR
activeData REF= ReferenceTarget;
SetBaseDatatypeReference();
END_METHOD

METHOD TryMakeReferenceTo : BOOL
VAR_INPUT
	Target : I_Datatype;
END_VAR
VAR
	pTargetData : POINTER TO ETcVnThresholdType;
END_VAR
IF NOT IsEquivalentTo(Target) THEN
	RETURN;
END_IF

pTargetData := Target.Address;
activeData REF= pTargetData^;
SetBaseDatatypeReference();
TryMakeReferenceTo := TRUE;
END_METHOD

PROPERTY PUBLIC Value : ETcVnThresholdType
GET
Value := activeData;
END_GET
SET
activeData := Value;
END_SET
END_PROPERTY

END_FUNCTION_BLOCK

// Datatypes/Enums/_ETcVnTimestamp
{attribute 'linkalways'} 
{attribute 'no_explicit_call' := 'This FB is a CLASS and must be accessed using methods or properties'}
{attribute 'enable_dynamic_creation'}
FUNCTION_BLOCK _ETcVnTimestamp EXTENDS EnumDatatypeBase
VAR
	localData : ETcVnTimestamp;
	activeData : REFERENCE TO ETcVnTimestamp;
	enumBaseDatatype : _ULINT(localData);
END_VAR

METHOD PROTECTED SetBaseDatatypeReference
VAR_INPUT
END_VAR
enumBaseDatatype.MakeReferenceTo(activeData);
END_METHOD

PROPERTY PUBLIC Address : PVOID
GET
Address := ADR(activeData);
END_GET
END_PROPERTY

METHOD PUBLIC ClearReference
VAR_INPUT
END_VAR
activeData REF= localData;
SetBaseDatatypeReference();
END_METHOD

PROPERTY PUBLIC Size : UDINT
GET
Size := SIZEOF(activeData);
END_GET
END_PROPERTY

METHOD FB_init : BOOL
VAR_INPUT
	bInitRetains : BOOL; // if TRUE, the retain variables are initialized (warm start / cold start)
	bInCopyCode : BOOL;  // if TRUE, the instance afterwards gets moved into the copy code (online change)
	InitialValue : ETcVnTimestamp;
END_VAR
localData := InitialValue;
AddBaseDatatype(enumBaseDatatype);
ClearReference();

AddLocalEnumeration('TCVN_TS_IMAGE_COMPLETED', ETcVnTimestamp.TCVN_TS_IMAGE_COMPLETED);
AddLocalEnumeration('TCVN_TS_RECEPTION_STARTED', ETcVnTimestamp.TCVN_TS_RECEPTION_STARTED);
AddLocalEnumeration('TCVN_TS_RECEPTION_FINISHED', ETcVnTimestamp.TCVN_TS_RECEPTION_FINISHED);
AddLocalEnumeration('TCVN_TS_GETCURRENTIMAGE', ETcVnTimestamp.TCVN_TS_GETCURRENTIMAGE);
AddLocalEnumeration('TCVN_TS_CAMERA', ETcVnTimestamp.TCVN_TS_CAMERA);
AddLocalEnumeration('TCVN_TS_CUSTOM', ETcVnTimestamp.TCVN_TS_CUSTOM);
AddLocalEnumeration('TCVN_TS_LAST_CHANGE', ETcVnTimestamp.TCVN_TS_LAST_CHANGE);
END_METHOD

METHOD PRIVATE AddLocalEnumeration
VAR_INPUT
	Enumeration : T_MAXSTRING;
	Value : ETcVnTimestamp;
END_VAR
AddEnumeration(Enumeration, Value);
END_METHOD

METHOD IsEnumeratorValueEqual : BOOL
VAR_INPUT
	Enumerator : I_KeyValueForwardEnumerator;
END_VAR
VAR
	storedValue : ETcVnTimestamp;
END_VAR
IF NOT Enumerator.TryGet(storedValue) THEN
	RETURN;
END_IF

IsEnumeratorValueEqual := storedValue = activeData;
END_METHOD

METHOD PUBLIC Clone : I_Datatype
VAR
    pClone : POINTER TO _ETcVnTimestamp;
END_VAR
pClone := __NEW(_ETcVnTimestamp(InitialValue := Value));
Clone := pClone^;
END_METHOD

PROPERTY PUBLIC Identifier : T_MAXSTRING
GET
Identifier := 'ETcVnTimestamp';
END_GET
END_PROPERTY

METHOD PUBLIC MakeReferenceTo
VAR_INPUT
	ReferenceTarget : REFERENCE TO ETcVnTimestamp;
END_VAR
activeData REF= ReferenceTarget;
SetBaseDatatypeReference();
END_METHOD

METHOD TryMakeReferenceTo : BOOL
VAR_INPUT
	Target : I_Datatype;
END_VAR
VAR
	pTargetData : POINTER TO ETcVnTimestamp;
END_VAR
IF NOT IsEquivalentTo(Target) THEN
	RETURN;
END_IF

pTargetData := Target.Address;
activeData REF= pTargetData^;
SetBaseDatatypeReference();
TryMakeReferenceTo := TRUE;
END_METHOD

PROPERTY PUBLIC Value : ETcVnTimestamp
GET
Value := activeData;
END_GET
SET
activeData := Value;
END_SET
END_PROPERTY

END_FUNCTION_BLOCK

// Datatypes/Enums/_ETcVnVectorCompareMethod
{attribute 'linkalways'} 
{attribute 'no_explicit_call' := 'This FB is a CLASS and must be accessed using methods or properties'}
{attribute 'enable_dynamic_creation'}
FUNCTION_BLOCK _ETcVnVectorCompareMethod EXTENDS EnumDatatypeBase
VAR
	localData : ETcVnVectorCompareMethod;
	activeData : REFERENCE TO ETcVnVectorCompareMethod;
	enumBaseDatatype : _DINT(localData);
END_VAR

METHOD PROTECTED SetBaseDatatypeReference
VAR_INPUT
END_VAR
enumBaseDatatype.MakeReferenceTo(activeData);
END_METHOD

PROPERTY PUBLIC Address : PVOID
GET
Address := ADR(activeData);
END_GET
END_PROPERTY

METHOD PUBLIC ClearReference
VAR_INPUT
END_VAR
activeData REF= localData;
SetBaseDatatypeReference();
END_METHOD

PROPERTY PUBLIC Size : UDINT
GET
Size := SIZEOF(activeData);
END_GET
END_PROPERTY

METHOD FB_init : BOOL
VAR_INPUT
	bInitRetains : BOOL; // if TRUE, the retain variables are initialized (warm start / cold start)
	bInCopyCode : BOOL;  // if TRUE, the instance afterwards gets moved into the copy code (online change)
	InitialValue : ETcVnVectorCompareMethod;
END_VAR
localData := InitialValue;
AddBaseDatatype(enumBaseDatatype);
ClearReference();

AddLocalEnumeration('TCVN_VCM_EUCLIDEAN', ETcVnVectorCompareMethod.TCVN_VCM_EUCLIDEAN);
AddLocalEnumeration('TCVN_VCM_ELEMENTWISE', ETcVnVectorCompareMethod.TCVN_VCM_ELEMENTWISE);
END_METHOD

METHOD PRIVATE AddLocalEnumeration
VAR_INPUT
	Enumeration : T_MAXSTRING;
	Value : ETcVnVectorCompareMethod;
END_VAR
AddEnumeration(Enumeration, Value);
END_METHOD

METHOD IsEnumeratorValueEqual : BOOL
VAR_INPUT
	Enumerator : I_KeyValueForwardEnumerator;
END_VAR
VAR
	storedValue : ETcVnVectorCompareMethod;
END_VAR
IF NOT Enumerator.TryGet(storedValue) THEN
	RETURN;
END_IF

IsEnumeratorValueEqual := storedValue = activeData;
END_METHOD

METHOD PUBLIC Clone : I_Datatype
VAR
    pClone : POINTER TO _ETcVnVectorCompareMethod;
END_VAR
pClone := __NEW(_ETcVnVectorCompareMethod(InitialValue := Value));
Clone := pClone^;
END_METHOD

PROPERTY PUBLIC Identifier : T_MAXSTRING
GET
Identifier := 'ETcVnVectorCompareMethod';
END_GET
END_PROPERTY

METHOD PUBLIC MakeReferenceTo
VAR_INPUT
	ReferenceTarget : REFERENCE TO ETcVnVectorCompareMethod;
END_VAR
activeData REF= ReferenceTarget;
SetBaseDatatypeReference();
END_METHOD

METHOD TryMakeReferenceTo : BOOL
VAR_INPUT
	Target : I_Datatype;
END_VAR
VAR
	pTargetData : POINTER TO ETcVnVectorCompareMethod;
END_VAR
IF NOT IsEquivalentTo(Target) THEN
	RETURN;
END_IF

pTargetData := Target.Address;
activeData REF= pTargetData^;
SetBaseDatatypeReference();
TryMakeReferenceTo := TRUE;
END_METHOD

PROPERTY PUBLIC Value : ETcVnVectorCompareMethod
GET
Value := activeData;
END_GET
SET
activeData := Value;
END_SET
END_PROPERTY

END_FUNCTION_BLOCK

// Datatypes/Enums/_ETcVnWorldCoordinateSystem
{attribute 'linkalways'} 
{attribute 'no_explicit_call' := 'This FB is a CLASS and must be accessed using methods or properties'}
{attribute 'enable_dynamic_creation'}
FUNCTION_BLOCK _ETcVnWorldCoordinateSystem EXTENDS EnumDatatypeBase
VAR
	localData : ETcVnWorldCoordinateSystem;
	activeData : REFERENCE TO ETcVnWorldCoordinateSystem;
	enumBaseDatatype : _DINT(localData);
END_VAR

METHOD PROTECTED SetBaseDatatypeReference
VAR_INPUT
END_VAR
enumBaseDatatype.MakeReferenceTo(activeData);
END_METHOD

PROPERTY PUBLIC Address : PVOID
GET
Address := ADR(activeData);
END_GET
END_PROPERTY

METHOD PUBLIC ClearReference
VAR_INPUT
END_VAR
activeData REF= localData;
SetBaseDatatypeReference();
END_METHOD

PROPERTY PUBLIC Size : UDINT
GET
Size := SIZEOF(activeData);
END_GET
END_PROPERTY

METHOD FB_init : BOOL
VAR_INPUT
	bInitRetains : BOOL; // if TRUE, the retain variables are initialized (warm start / cold start)
	bInCopyCode : BOOL;  // if TRUE, the instance afterwards gets moved into the copy code (online change)
	InitialValue : ETcVnWorldCoordinateSystem;
END_VAR
localData := InitialValue;
AddBaseDatatype(enumBaseDatatype);
ClearReference();

AddLocalEnumeration('TCVN_WCS_X_RIGHT_Y_DOWN' , ETcVnWorldCoordinateSystem.TCVN_WCS_X_RIGHT_Y_DOWN);
AddLocalEnumeration('TCVN_WCS_X_DOWN_Y_RIGHT', ETcVnWorldCoordinateSystem.TCVN_WCS_X_DOWN_Y_RIGHT);
AddLocalEnumeration('TCVN_WCS_X_LEFT_Y_DOWN', ETcVnWorldCoordinateSystem.TCVN_WCS_X_LEFT_Y_DOWN);
AddLocalEnumeration('TCVN_WCS_X_UP_Y_RIGHT', ETcVnWorldCoordinateSystem.TCVN_WCS_X_UP_Y_RIGHT);
AddLocalEnumeration('TCVN_WCS_X_RIGHT_Y_UP', ETcVnWorldCoordinateSystem.TCVN_WCS_X_RIGHT_Y_UP);
AddLocalEnumeration('TCVN_WCS_X_DOWN_Y_LEFT', ETcVnWorldCoordinateSystem.TCVN_WCS_X_DOWN_Y_LEFT);
AddLocalEnumeration('TCVN_WCS_X_LEFT_Y_UP', ETcVnWorldCoordinateSystem.TCVN_WCS_X_LEFT_Y_UP);
AddLocalEnumeration('TCVN_WCS_X_UP_Y_LEFT', ETcVnWorldCoordinateSystem.TCVN_WCS_X_UP_Y_LEFT);
END_METHOD

METHOD PRIVATE AddLocalEnumeration
VAR_INPUT
	Enumeration : T_MAXSTRING;
	Value : ETcVnWorldCoordinateSystem;
END_VAR
AddEnumeration(Enumeration, Value);
END_METHOD

METHOD IsEnumeratorValueEqual : BOOL
VAR_INPUT
	Enumerator : I_KeyValueForwardEnumerator;
END_VAR
VAR
	storedValue : ETcVnWorldCoordinateSystem;
END_VAR
IF NOT Enumerator.TryGet(storedValue) THEN
	RETURN;
END_IF

IsEnumeratorValueEqual := storedValue = activeData;
END_METHOD

METHOD PUBLIC Clone : I_Datatype
VAR
    pClone : POINTER TO _ETcVnWorldCoordinateSystem;
END_VAR
pClone := __NEW(_ETcVnWorldCoordinateSystem(InitialValue := Value));
Clone := pClone^;
END_METHOD

PROPERTY PUBLIC Identifier : T_MAXSTRING
GET
Identifier := 'ETcVnWorldCoordinateSystem';
END_GET
END_PROPERTY

METHOD PUBLIC MakeReferenceTo
VAR_INPUT
	ReferenceTarget : REFERENCE TO ETcVnWorldCoordinateSystem;
END_VAR
activeData REF= ReferenceTarget;
SetBaseDatatypeReference();
END_METHOD

METHOD TryMakeReferenceTo : BOOL
VAR_INPUT
	Target : I_Datatype;
END_VAR
VAR
	pTargetData : POINTER TO ETcVnWorldCoordinateSystem;
END_VAR
IF NOT IsEquivalentTo(Target) THEN
	RETURN;
END_IF

pTargetData := Target.Address;
activeData REF= pTargetData^;
SetBaseDatatypeReference();
TryMakeReferenceTo := TRUE;
END_METHOD

PROPERTY PUBLIC Value : ETcVnWorldCoordinateSystem
GET
Value := activeData;
END_GET
SET
activeData := Value;
END_SET
END_PROPERTY

END_FUNCTION_BLOCK

// Datatypes/Enums/_ETcWatchdogAccumulationType
{attribute 'linkalways'} 
{attribute 'no_explicit_call' := 'This FB is a CLASS and must be accessed using methods or properties'}
{attribute 'enable_dynamic_creation'}
FUNCTION_BLOCK _ETcWatchdogAccumulationType EXTENDS EnumDatatypeBase
VAR
	localData : ETcWatchdogAccumulationType;
	activeData : REFERENCE TO ETcWatchdogAccumulationType;
	enumBaseDatatype : _UINT(localData);
END_VAR

METHOD PROTECTED SetBaseDatatypeReference
VAR_INPUT
END_VAR
enumBaseDatatype.MakeReferenceTo(activeData);
END_METHOD

PROPERTY PUBLIC Address : PVOID
GET
Address := ADR(activeData);
END_GET
END_PROPERTY

METHOD PUBLIC ClearReference
VAR_INPUT
END_VAR
activeData REF= localData;
SetBaseDatatypeReference();
END_METHOD

PROPERTY PUBLIC Size : UDINT
GET
Size := SIZEOF(activeData);
END_GET
END_PROPERTY

METHOD FB_init : BOOL
VAR_INPUT
	bInitRetains : BOOL; // if TRUE, the retain variables are initialized (warm start / cold start)
	bInCopyCode : BOOL;  // if TRUE, the instance afterwards gets moved into the copy code (online change)
	InitialValue : ETcWatchdogAccumulationType;
END_VAR
localData := InitialValue;
AddBaseDatatype(enumBaseDatatype);
ClearReference();

AddLocalEnumeration('WD_ACC_TYPE_MEAN', ETcWatchdogAccumulationType.WD_ACC_TYPE_MEAN);
AddLocalEnumeration('WD_ACC_TYPE_PRODUCT', ETcWatchdogAccumulationType.WD_ACC_TYPE_PRODUCT);
END_METHOD

METHOD PRIVATE AddLocalEnumeration
VAR_INPUT
	Enumeration : T_MAXSTRING;
	Value : ETcWatchdogAccumulationType;
END_VAR
AddEnumeration(Enumeration, Value);
END_METHOD

METHOD IsEnumeratorValueEqual : BOOL
VAR_INPUT
	Enumerator : I_KeyValueForwardEnumerator;
END_VAR
VAR
	storedValue : ETcWatchdogAccumulationType;
END_VAR
IF NOT Enumerator.TryGet(storedValue) THEN
	RETURN;
END_IF

IsEnumeratorValueEqual := storedValue = activeData;
END_METHOD

METHOD PUBLIC Clone : I_Datatype
VAR
    pClone : POINTER TO _ETcWatchdogAccumulationType;
END_VAR
pClone := __NEW(_ETcWatchdogAccumulationType(InitialValue := Value));
Clone := pClone^;
END_METHOD

PROPERTY PUBLIC Identifier : T_MAXSTRING
GET
Identifier := 'ETcWatchdogAccumulationType';
END_GET
END_PROPERTY

METHOD PUBLIC MakeReferenceTo
VAR_INPUT
	ReferenceTarget : REFERENCE TO ETcWatchdogAccumulationType;
END_VAR
activeData REF= ReferenceTarget;
SetBaseDatatypeReference();
END_METHOD

METHOD TryMakeReferenceTo : BOOL
VAR_INPUT
	Target : I_Datatype;
END_VAR
VAR
	pTargetData : POINTER TO ETcWatchdogAccumulationType;
END_VAR
IF NOT IsEquivalentTo(Target) THEN
	RETURN;
END_IF

pTargetData := Target.Address;
activeData REF= pTargetData^;
SetBaseDatatypeReference();
TryMakeReferenceTo := TRUE;
END_METHOD

PROPERTY PUBLIC Value : ETcWatchdogAccumulationType
GET
Value := activeData;
END_GET
SET
activeData := Value;
END_SET
END_PROPERTY

END_FUNCTION_BLOCK

// Datatypes/Enums/_GEV_CAMERA_STATE
{attribute 'linkalways'} 
{attribute 'no_explicit_call' := 'This FB is a CLASS and must be accessed using methods or properties'}
{attribute 'enable_dynamic_creation'}
FUNCTION_BLOCK _GEV_CAMERA_STATE EXTENDS EnumDatatypeBase
VAR
	localData : GEV_CAMERA_STATE;
	activeData : REFERENCE TO GEV_CAMERA_STATE;
	enumBaseDatatype : _BYTE(localData);
END_VAR

METHOD PROTECTED SetBaseDatatypeReference
VAR_INPUT
END_VAR
enumBaseDatatype.MakeReferenceTo(activeData);
END_METHOD

PROPERTY PUBLIC Address : PVOID
GET
Address := ADR(activeData);
END_GET
END_PROPERTY

METHOD PUBLIC ClearReference
VAR_INPUT
END_VAR
activeData REF= localData;
SetBaseDatatypeReference();
END_METHOD

PROPERTY PUBLIC Size : UDINT
GET
Size := SIZEOF(activeData);
END_GET
END_PROPERTY

METHOD FB_init : BOOL
VAR_INPUT
	bInitRetains : BOOL; // if TRUE, the retain variables are initialized (warm start / cold start)
	bInCopyCode : BOOL;  // if TRUE, the instance afterwards gets moved into the copy code (online change)
	InitialValue : GEV_CAMERA_STATE;
END_VAR
localData := InitialValue;
AddBaseDatatype(enumBaseDatatype);
ClearReference();

AddLocalEnumeration('GEV_CAMERA_IDLE', GEV_CAMERA_STATE.GEV_CAMERA_IDLE);
AddLocalEnumeration('GEV_CONTROL_CHANNEL_OPEN_MASK', GEV_CAMERA_STATE.GEV_CONTROL_CHANNEL_OPEN_MASK);
AddLocalEnumeration('GEV_STREAM_CHANNELS_OPEN_MASK', GEV_CAMERA_STATE.GEV_STREAM_CHANNELS_OPEN_MASK);
AddLocalEnumeration('GEV_CONTROL_CHANNEL_OPEN', GEV_CAMERA_STATE.GEV_CONTROL_CHANNEL_OPEN);
AddLocalEnumeration('GEV_STREAM_CHANNELS_OPEN', GEV_CAMERA_STATE.GEV_STREAM_CHANNELS_OPEN);
END_METHOD

METHOD PRIVATE AddLocalEnumeration
VAR_INPUT
	Enumeration : T_MAXSTRING;
	Value : GEV_CAMERA_STATE;
END_VAR
AddEnumeration(Enumeration, Value);
END_METHOD

METHOD IsEnumeratorValueEqual : BOOL
VAR_INPUT
	Enumerator : I_KeyValueForwardEnumerator;
END_VAR
VAR
	storedValue : GEV_CAMERA_STATE;
END_VAR
IF NOT Enumerator.TryGet(storedValue) THEN
	RETURN;
END_IF

IsEnumeratorValueEqual := storedValue = activeData;
END_METHOD

METHOD PUBLIC Clone : I_Datatype
VAR
    pClone : POINTER TO _GEV_CAMERA_STATE;
END_VAR
pClone := __NEW(_GEV_CAMERA_STATE(InitialValue := Value));
Clone := pClone^;
END_METHOD

PROPERTY PUBLIC Identifier : T_MAXSTRING
GET
Identifier := 'GEV_CAMERA_STATE';
END_GET
END_PROPERTY

METHOD PUBLIC MakeReferenceTo
VAR_INPUT
	ReferenceTarget : REFERENCE TO GEV_CAMERA_STATE;
END_VAR
activeData REF= ReferenceTarget;
SetBaseDatatypeReference();
END_METHOD

METHOD TryMakeReferenceTo : BOOL
VAR_INPUT
	Target : I_Datatype;
END_VAR
VAR
	pTargetData : POINTER TO GEV_CAMERA_STATE;
END_VAR
IF NOT IsEquivalentTo(Target) THEN
	RETURN;
END_IF

pTargetData := Target.Address;
activeData REF= pTargetData^;
SetBaseDatatypeReference();
TryMakeReferenceTo := TRUE;
END_METHOD

PROPERTY PUBLIC Value : GEV_CAMERA_STATE
GET
Value := activeData;
END_GET
SET
activeData := Value;
END_SET
END_PROPERTY

END_FUNCTION_BLOCK

// Datatypes/Interfaces/Containers/ITcVnContainer/_ITcVnContainer
{attribute 'linkalways'} 
{attribute 'no_explicit_call' := 'This FB is a CLASS and must be accessed using methods or properties'}
{attribute 'enable_dynamic_creation'}
FUNCTION_BLOCK _ITcVnContainer EXTENDS InterfaceDatatypeBase IMPLEMENTS I_InterfaceDatatype_ITcVnContainer
VAR
	localData : ITcVnContainer;
	activeData : REFERENCE TO ITcVnContainer REF= localData;
END_VAR

PROPERTY PUBLIC Address : PVOID
GET
Address := ADR(activeData);
END_GET
END_PROPERTY

METHOD PUBLIC ClearReference
VAR_INPUT
END_VAR
activeData REF= localData;
END_METHOD

PROPERTY PUBLIC Size : UDINT
GET
Size := SIZEOF(activeData);
END_GET
END_PROPERTY

METHOD FB_exit : BOOL
VAR_INPUT
	bInCopyCode : BOOL; // if TRUE, the exit method is called for exiting an instance that is copied afterwards (online change).
END_VAR
IF bInCopyCode THEN
	RETURN;
END_IF

TryTcReleaseLocal();
END_METHOD

METHOD PRIVATE Serialize_ContainerType_String_SINT
VAR_INPUT
	Serializer : I_Serializer;
	TargetContainer : ITcVnContainer;
END_VAR
VAR
	hr : HRESULT;
	_value : _STRING('');
END_VAR
hr := F_VN_ExportContainer_String(TargetContainer, _value.Value, SIZEOF(_value.Value), S_OK);
Serializer.StartArray();

IF SUCCEEDED(hr) THEN
	Serializer.AddObject(_value);
ELSE
	Serializer.AddNull();
END_IF

Serializer.EndArray();
END_METHOD

METHOD PRIVATE Serialize_ContainerType_Vector_DINT
VAR_INPUT
	Serializer : I_Serializer;
	TargetContainer : ITcVnContainer;
END_VAR
VAR
	hr : HRESULT;
	_value : _DINT(0);
	elementCount : ULINT;
	i : ULINT;
END_VAR
TargetContainer.GetElementNum(elementCount);
Serializer.StartArray();

IF elementCount > 0 THEN
	FOR i := 0 TO elementCount - 1 DO 
		
		hr := F_VN_GetAt_DINT(TargetContainer, _value.Value, i, S_OK);
		
		IF SUCCEEDED(hr) THEN
			Serializer.AddObject(_value);
		ELSE
			Serializer.AddNull();
		END_IF
		
	END_FOR
END_IF

Serializer.EndArray();
END_METHOD

METHOD PRIVATE Serialize_ContainerType_Vector_INT
VAR_INPUT
	Serializer : I_Serializer;
	TargetContainer : ITcVnContainer;
END_VAR
VAR
	hr : HRESULT;
	_value : _INT(0);
	elementCount : ULINT;
	i : ULINT;
END_VAR
TargetContainer.GetElementNum(elementCount);
Serializer.StartArray();

IF elementCount > 0 THEN
	FOR i := 0 TO elementCount - 1 DO 
		
		hr := F_VN_GetAt_INT(TargetContainer, _value.Value, i, S_OK);
		
		IF SUCCEEDED(hr) THEN
			Serializer.AddObject(_value);
		ELSE
			Serializer.AddNull();
		END_IF
		
	END_FOR
END_IF

Serializer.EndArray();
END_METHOD

METHOD PRIVATE Serialize_ContainerType_Vector_ITcVnImage
VAR_INPUT
	Serializer : I_Serializer;
	TargetContainer : ITcVnContainer;
END_VAR
VAR
	hr : HRESULT;
	_value : _ITcVnImage;
	elementCount : ULINT;
	i : ULINT;
END_VAR
TargetContainer.GetElementNum(elementCount);
Serializer.StartArray();

IF elementCount > 0 THEN
	FOR i := 0 TO elementCount - 1 DO 
		
		hr := F_VN_GetAt_ITcVnImage(TargetContainer, _value.Value, i, S_OK);
		
		IF SUCCEEDED(hr) THEN
			Serializer.AddObject(_value);
		ELSE
			Serializer.AddNull();
		END_IF
	
	END_FOR
END_IF

IF _value.Value <> 0 THEN
	_value.Value.TcRelease();
END_IF

Serializer.EndArray();
END_METHOD

METHOD PRIVATE Serialize_ContainerType_Vector_LREAL
VAR_INPUT
	Serializer : I_Serializer;
	TargetContainer : ITcVnContainer;
END_VAR
VAR
	hr : HRESULT;
	_value : _LREAL(0);
	elementCount : ULINT;
	i : ULINT;
END_VAR
TargetContainer.GetElementNum(elementCount);
Serializer.StartArray();

IF elementCount > 0 THEN
	FOR i := 0 TO elementCount - 1 DO 
		
		hr := F_VN_GetAt_LREAL(TargetContainer, _value.Value, i, S_OK);
		
		IF SUCCEEDED(hr) THEN
			Serializer.AddObject(_value);
		ELSE
			Serializer.AddNull();
		END_IF
		
	END_FOR
END_IF

Serializer.EndArray();
END_METHOD

METHOD PRIVATE Serialize_ContainerType_Vector_REAL
VAR_INPUT
	Serializer : I_Serializer;
	TargetContainer : ITcVnContainer;
END_VAR
VAR
	hr : HRESULT;
	_value : _REAL(0);
	elementCount : ULINT;
	i : ULINT;
END_VAR
TargetContainer.GetElementNum(elementCount);
Serializer.StartArray();

IF elementCount > 0 THEN
	FOR i := 0 TO elementCount - 1 DO 
		
		hr := F_VN_GetAt_REAL(TargetContainer, _value.Value, i, S_OK);
		
		IF SUCCEEDED(hr) THEN
			Serializer.AddObject(_value);
		ELSE
			Serializer.AddNull();
		END_IF
		
	END_FOR
END_IF

Serializer.EndArray();
END_METHOD

METHOD PRIVATE Serialize_ContainerType_Vector_SINT
VAR_INPUT
	Serializer : I_Serializer;
	TargetContainer : ITcVnContainer;
END_VAR
VAR
	hr : HRESULT;
	_value : _SINT(0);
	elementCount : ULINT;
	i : ULINT;
END_VAR
TargetContainer.GetElementNum(elementCount);
Serializer.StartArray();

IF elementCount > 0 THEN
	FOR i := 0 TO elementCount - 1 DO 
		
		hr := F_VN_GetAt_SINT(TargetContainer, _value.Value, i, S_OK);
		
		IF SUCCEEDED(hr) THEN
			Serializer.AddObject(_value);
		ELSE
			Serializer.AddNull();
		END_IF
		
	END_FOR
END_IF

Serializer.EndArray();
END_METHOD

METHOD PRIVATE Serialize_ContainerType_Vector_String_SINT
VAR_INPUT
	Serializer : I_Serializer;
	TargetContainer : ITcVnContainer;
END_VAR
VAR
	hr : HRESULT;
	_value : _STRING('');
	elementCount : ULINT;
	i : ULINT;
END_VAR
TargetContainer.GetElementNum(elementCount);
Serializer.StartArray();

IF elementCount > 0 THEN
	FOR i := 0 TO elementCount - 1 DO 
		
		hr := F_VN_ExportSubContainer_String(TargetContainer, i, _value.Value, SIZEOF(_value.Value), S_OK);
		
		IF SUCCEEDED(hr) THEN
			Serializer.AddObject(_value);
		ELSE
			Serializer.AddNull();
		END_IF
		
	END_FOR
END_IF

Serializer.EndArray();
END_METHOD

METHOD PRIVATE Serialize_ContainerType_Vector_TcVnDMatch
VAR_INPUT
	Serializer : I_Serializer;
	TargetContainer : ITcVnContainer;
END_VAR
VAR
	hr : HRESULT;
	_value : _TcVnDMatch();
	elementCount : ULINT;
	i : ULINT;
END_VAR
TargetContainer.GetElementNum(elementCount);
Serializer.StartArray();

IF elementCount > 0 THEN
	FOR i := 0 TO elementCount - 1 DO 
		
		hr := F_VN_GetAt_TcVnDMatch(TargetContainer, _value.Value, i, S_OK);
		
		IF SUCCEEDED(hr) THEN
			Serializer.AddObject(_value);
		ELSE
			Serializer.AddNull();
		END_IF
		
	END_FOR
END_IF

Serializer.EndArray();
END_METHOD

METHOD PRIVATE Serialize_ContainerType_Vector_TcVnKeyPoint
VAR_INPUT
	Serializer : I_Serializer;
	TargetContainer : ITcVnContainer;
END_VAR
VAR
	hr : HRESULT;
	_value : _TcVnKeyPoint();
	elementCount : ULINT;
	i : ULINT;
END_VAR
TargetContainer.GetElementNum(elementCount);
Serializer.StartArray();

IF elementCount > 0 THEN
	FOR i := 0 TO elementCount - 1 DO 
		
		hr := F_VN_GetAt_TcVnKeyPoint(TargetContainer, _value.Value, i, S_OK);
		
		IF SUCCEEDED(hr) THEN
			Serializer.AddObject(_value);
		ELSE
			Serializer.AddNull();
		END_IF
		
	END_FOR
END_IF

Serializer.EndArray();
END_METHOD

METHOD PRIVATE Serialize_ContainerType_Vector_TcVnPoint2_DINT
VAR_INPUT
	Serializer : I_Serializer;
	TargetContainer : ITcVnContainer;
END_VAR
VAR
	hr : HRESULT;
	_value : _TcVnPoint2_DINT();
	elementCount : ULINT;
	i : ULINT;
END_VAR
TargetContainer.GetElementNum(elementCount);
Serializer.StartArray();

IF elementCount > 0 THEN
	FOR i := 0 TO elementCount - 1 DO 
		
		hr := F_VN_GetAt_TcVnPoint2_DINT (TargetContainer, _value.Value, i, S_OK);
		
		IF SUCCEEDED(hr) THEN
			Serializer.AddObject(_value);
		ELSE
			Serializer.AddNull();
		END_IF
		
	END_FOR
END_IF

Serializer.EndArray();
END_METHOD

METHOD PRIVATE Serialize_ContainerType_Vector_TcVnPoint2_LREAL
VAR_INPUT
	Serializer : I_Serializer;
	TargetContainer : ITcVnContainer;
END_VAR
VAR
	hr : HRESULT;
	_value : _TcVnPoint2_LREAL();
	elementCount : ULINT;
	i : ULINT;
END_VAR
TargetContainer.GetElementNum(elementCount);
Serializer.StartArray();

IF elementCount > 0 THEN
	FOR i := 0 TO elementCount - 1 DO 
		
		hr := F_VN_GetAt_TcVnPoint2_LREAL (TargetContainer, _value.Value, i, S_OK);
		
		IF SUCCEEDED(hr) THEN
			Serializer.AddObject(_value);
		ELSE
			Serializer.AddNull();
		END_IF
		
	END_FOR
END_IF

Serializer.EndArray();
END_METHOD

METHOD PRIVATE Serialize_ContainerType_Vector_TcVnPoint2_REAL
VAR_INPUT
	Serializer : I_Serializer;
	TargetContainer : ITcVnContainer;
END_VAR
VAR
	hr : HRESULT;
	_value : _TcVnPoint2_REAL();
	elementCount : ULINT;
	i : ULINT;
END_VAR
TargetContainer.GetElementNum(elementCount);
Serializer.StartArray();

IF elementCount > 0 THEN
	FOR i := 0 TO elementCount - 1 DO 
		
		hr := F_VN_GetAt_TcVnPoint2_REAL (TargetContainer, _value.Value, i, S_OK);
		
		IF SUCCEEDED(hr) THEN
			Serializer.AddObject(_value);
		ELSE
			Serializer.AddNull();
		END_IF
		
	END_FOR
END_IF

Serializer.EndArray();
END_METHOD

METHOD PRIVATE Serialize_ContainerType_Vector_TcVnPoint3_LREAL
VAR_INPUT
	Serializer : I_Serializer;
	TargetContainer : ITcVnContainer;
END_VAR
VAR
	hr : HRESULT;
	_value : _TcVnPoint3_LREAL();
	elementCount : ULINT;
	i : ULINT;
END_VAR
TargetContainer.GetElementNum(elementCount);
Serializer.StartArray();

IF elementCount > 0 THEN
	FOR i := 0 TO elementCount - 1 DO 
		
		hr := F_VN_GetAt_TcVnPoint3_LREAL (TargetContainer, _value.Value, i, S_OK);
		
		IF SUCCEEDED(hr) THEN
			Serializer.AddObject(_value);
		ELSE
			Serializer.AddNull();
		END_IF
		
	END_FOR
END_IF

Serializer.EndArray();
END_METHOD

METHOD PRIVATE Serialize_ContainerType_Vector_TcVnPoint3_REAL
VAR_INPUT
	Serializer : I_Serializer;
	TargetContainer : ITcVnContainer;
END_VAR
VAR
	hr : HRESULT;
	_value : _TcVnPoint3_REAL();
	elementCount : ULINT;
	i : ULINT;
END_VAR
TargetContainer.GetElementNum(elementCount);
Serializer.StartArray();

IF elementCount > 0 THEN
	FOR i := 0 TO elementCount - 1 DO 
		
		hr := F_VN_GetAt_TcVnPoint3_REAL (TargetContainer, _value.Value, i, S_OK);
		
		IF SUCCEEDED(hr) THEN
			Serializer.AddObject(_value);
		ELSE
			Serializer.AddNull();
		END_IF
		
	END_FOR
END_IF

Serializer.EndArray();
END_METHOD

METHOD PRIVATE Serialize_ContainerType_Vector_TcVnRectangle_DINT
VAR_INPUT
	Serializer : I_Serializer;
	TargetContainer : ITcVnContainer;
END_VAR
VAR
	hr : HRESULT;
	_value : _TcVnRectangle_DINT();
	elementCount : ULINT;
	i : ULINT;
END_VAR
TargetContainer.GetElementNum(elementCount);
Serializer.StartArray();

IF elementCount > 0 THEN
	FOR i := 0 TO elementCount - 1 DO 
		
		hr := F_VN_GetAt_TcVnRectangle_DINT(TargetContainer, _value.Value, i, S_OK);
		
		IF SUCCEEDED(hr) THEN
			Serializer.AddObject(_value);
		ELSE
			Serializer.AddNull();
		END_IF
		
	END_FOR
END_IF

Serializer.EndArray();
END_METHOD

METHOD PRIVATE Serialize_ContainerType_Vector_TcVnRotatedRectangle
VAR_INPUT
	Serializer : I_Serializer;
	TargetContainer : ITcVnContainer;
END_VAR
VAR
	hr : HRESULT;
	_value : _TcVnRotatedRectangle();
	elementCount : ULINT;
	i : ULINT;
END_VAR
TargetContainer.GetElementNum(elementCount);
Serializer.StartArray();

IF elementCount > 0 THEN
	FOR i := 0 TO elementCount - 1 DO 
		
		hr := F_VN_GetAt_TcVnRotatedRectangle(TargetContainer, _value.Value, i, S_OK);
		
		IF SUCCEEDED(hr) THEN
			Serializer.AddObject(_value);
		ELSE
			Serializer.AddNull();
		END_IF
		
	END_FOR
END_IF

Serializer.EndArray();
END_METHOD

METHOD PRIVATE Serialize_ContainerType_Vector_TcVnVector2_DINT
VAR_INPUT
	Serializer : I_Serializer;
	TargetContainer : ITcVnContainer;
END_VAR
VAR
	hr : HRESULT;
	_value : _TcVnVector2_DINT();
	elementCount : ULINT;
	i : ULINT;
END_VAR
TargetContainer.GetElementNum(elementCount);
Serializer.StartArray();

IF elementCount > 0 THEN
	FOR i := 0 TO elementCount - 1 DO 
		
		hr := F_VN_GetAt_TcVnVector2_DINT(TargetContainer, _value.Value, i, S_OK);
		
		IF SUCCEEDED(hr) THEN
			Serializer.AddObject(_value);
		ELSE
			Serializer.AddNull();
		END_IF
		
	END_FOR
END_IF

Serializer.EndArray();
END_METHOD

METHOD PRIVATE Serialize_ContainerType_Vector_TcVnVector2_INT
VAR_INPUT
	Serializer : I_Serializer;
	TargetContainer : ITcVnContainer;
END_VAR
VAR
	hr : HRESULT;
	_value : _TcVnVector2_INT();
	elementCount : ULINT;
	i : ULINT;
END_VAR
TargetContainer.GetElementNum(elementCount);
Serializer.StartArray();

IF elementCount > 0 THEN
	FOR i := 0 TO elementCount - 1 DO 
		
		hr := F_VN_GetAt_TcVnVector2_INT(TargetContainer, _value.Value, i, S_OK);
		
		IF SUCCEEDED(hr) THEN
			Serializer.AddObject(_value);
		ELSE
			Serializer.AddNull();
		END_IF
		
	END_FOR
END_IF

Serializer.EndArray();
END_METHOD

METHOD PRIVATE Serialize_ContainerType_Vector_TcVnVector2_REAL
VAR_INPUT
	Serializer : I_Serializer;
	TargetContainer : ITcVnContainer;
END_VAR
VAR
	hr : HRESULT;
	_value : _TcVnVector2_REAL();
	elementCount : ULINT;
	i : ULINT;
END_VAR
TargetContainer.GetElementNum(elementCount);
Serializer.StartArray();

IF elementCount > 0 THEN
	FOR i := 0 TO elementCount - 1 DO 
		
		hr := F_VN_GetAt_TcVnVector2_REAL(TargetContainer, _value.Value, i, S_OK);
		
		IF SUCCEEDED(hr) THEN
			Serializer.AddObject(_value);
		ELSE
			Serializer.AddNull();
		END_IF
		
	END_FOR
END_IF

Serializer.EndArray();
END_METHOD

METHOD PRIVATE Serialize_ContainerType_Vector_TcVnVector2_SINT
VAR_INPUT
	Serializer : I_Serializer;
	TargetContainer : ITcVnContainer;
END_VAR
VAR
	hr : HRESULT;
	_value : _TcVnVector2_SINT();
	elementCount : ULINT;
	i : ULINT;
END_VAR
TargetContainer.GetElementNum(elementCount);
Serializer.StartArray();

IF elementCount > 0 THEN
	FOR i := 0 TO elementCount - 1 DO 
		
		hr := F_VN_GetAt_TcVnVector2_SINT(TargetContainer, _value.Value, i, S_OK);
		
		IF SUCCEEDED(hr) THEN
			Serializer.AddObject(_value);
		ELSE
			Serializer.AddNull();
		END_IF
		
	END_FOR
END_IF

Serializer.EndArray();
END_METHOD

METHOD PRIVATE Serialize_ContainerType_Vector_TcVnVector2_UINT
VAR_INPUT
	Serializer : I_Serializer;
	TargetContainer : ITcVnContainer;
END_VAR
VAR
	hr : HRESULT;
	_value : _TcVnVector2_UINT();
	elementCount : ULINT;
	i : ULINT;
END_VAR
TargetContainer.GetElementNum(elementCount);
Serializer.StartArray();

IF elementCount > 0 THEN
	FOR i := 0 TO elementCount - 1 DO 
		
		hr := F_VN_GetAt_TcVnVector2_UINT(TargetContainer, _value.Value, i, S_OK);
		
		IF SUCCEEDED(hr) THEN
			Serializer.AddObject(_value);
		ELSE
			Serializer.AddNull();
		END_IF
		
	END_FOR
END_IF

Serializer.EndArray();
END_METHOD

METHOD PRIVATE Serialize_ContainerType_Vector_TcVnVector2_USINT
VAR_INPUT
	Serializer : I_Serializer;
	TargetContainer : ITcVnContainer;
END_VAR
VAR
	hr : HRESULT;
	_value : _TcVnVector2_USINT();
	elementCount : ULINT;
	i : ULINT;
END_VAR
TargetContainer.GetElementNum(elementCount);
Serializer.StartArray();

IF elementCount > 0 THEN
	FOR i := 0 TO elementCount - 1 DO 
		
		hr := F_VN_GetAt_TcVnVector2_USINT(TargetContainer, _value.Value, i, S_OK);
		
		IF SUCCEEDED(hr) THEN
			Serializer.AddObject(_value);
		ELSE
			Serializer.AddNull();
		END_IF
		
	END_FOR
END_IF

Serializer.EndArray();
END_METHOD

METHOD PRIVATE Serialize_ContainerType_Vector_TcVnVector3_INT
VAR_INPUT
	Serializer : I_Serializer;
	TargetContainer : ITcVnContainer;
END_VAR
VAR
	hr : HRESULT;
	_value : _TcVnVector3_INT();
	elementCount : ULINT;
	i : ULINT;
END_VAR
TargetContainer.GetElementNum(elementCount);
Serializer.StartArray();

IF elementCount > 0 THEN
	FOR i := 0 TO elementCount - 1 DO 
		
		hr := F_VN_GetAt_TcVnVector3_INT(TargetContainer, _value.Value, i, S_OK);
		
		IF SUCCEEDED(hr) THEN
			Serializer.AddObject(_value);
		ELSE
			Serializer.AddNull();
		END_IF
		
	END_FOR
END_IF

Serializer.EndArray();
END_METHOD

METHOD PRIVATE Serialize_ContainerType_Vector_TcVnVector3_REAL
VAR_INPUT
	Serializer : I_Serializer;
	TargetContainer : ITcVnContainer;
END_VAR
VAR
	hr : HRESULT;
	_value : _TcVnVector3_REAL();
	elementCount : ULINT;
	i : ULINT;
END_VAR
TargetContainer.GetElementNum(elementCount);
Serializer.StartArray();

IF elementCount > 0 THEN
	FOR i := 0 TO elementCount - 1 DO 
		
		hr := F_VN_GetAt_TcVnVector3_REAL(TargetContainer, _value.Value, i, S_OK);
		
		IF SUCCEEDED(hr) THEN
			Serializer.AddObject(_value);
		ELSE
			Serializer.AddNull();
		END_IF
		
	END_FOR
END_IF

Serializer.EndArray();
END_METHOD

METHOD PRIVATE Serialize_ContainerType_Vector_TcVnVector3_SINT
VAR_INPUT
	Serializer : I_Serializer;
	TargetContainer : ITcVnContainer;
END_VAR
VAR
	hr : HRESULT;
	_value : _TcVnVector3_SINT();
	elementCount : ULINT;
	i : ULINT;
END_VAR
TargetContainer.GetElementNum(elementCount);
Serializer.StartArray();

IF elementCount > 0 THEN
	FOR i := 0 TO elementCount - 1 DO 
		
		hr := F_VN_GetAt_TcVnVector3_SINT(TargetContainer, _value.Value, i, S_OK);
		
		IF SUCCEEDED(hr) THEN
			Serializer.AddObject(_value);
		ELSE
			Serializer.AddNull();
		END_IF
		
	END_FOR
END_IF

Serializer.EndArray();
END_METHOD

METHOD PRIVATE Serialize_ContainerType_Vector_TcVnVector3_UINT
VAR_INPUT
	Serializer : I_Serializer;
	TargetContainer : ITcVnContainer;
END_VAR
VAR
	hr : HRESULT;
	_value : _TcVnVector3_UINT();
	elementCount : ULINT;
	i : ULINT;
END_VAR
TargetContainer.GetElementNum(elementCount);
Serializer.StartArray();

IF elementCount > 0 THEN
	FOR i := 0 TO elementCount - 1 DO 
		
		hr := F_VN_GetAt_TcVnVector3_UINT(TargetContainer, _value.Value, i, S_OK);
		
		IF SUCCEEDED(hr) THEN
			Serializer.AddObject(_value);
		ELSE
			Serializer.AddNull();
		END_IF
		
	END_FOR
END_IF

Serializer.EndArray();
END_METHOD

METHOD PRIVATE Serialize_ContainerType_Vector_TcVnVector3_USINT
VAR_INPUT
	Serializer : I_Serializer;
	TargetContainer : ITcVnContainer;
END_VAR
VAR
	hr : HRESULT;
	_value : _TcVnVector3_USINT();
	elementCount : ULINT;
	i : ULINT;
END_VAR
TargetContainer.GetElementNum(elementCount);
Serializer.StartArray();

IF elementCount > 0 THEN
	FOR i := 0 TO elementCount - 1 DO 
		
		hr := F_VN_GetAt_TcVnVector3_USINT(TargetContainer, _value.Value, i, S_OK);
		
		IF SUCCEEDED(hr) THEN
			Serializer.AddObject(_value);
		ELSE
			Serializer.AddNull();
		END_IF
		
	END_FOR
END_IF

Serializer.EndArray();
END_METHOD

METHOD PRIVATE Serialize_ContainerType_Vector_TcVnVector4_DINT
VAR_INPUT
	Serializer : I_Serializer;
	TargetContainer : ITcVnContainer;
END_VAR
VAR
	hr : HRESULT;
	_value : _TcVnVector4_DINT();
	elementCount : ULINT;
	i : ULINT;
END_VAR
TargetContainer.GetElementNum(elementCount);
Serializer.StartArray();

IF elementCount > 0 THEN
	FOR i := 0 TO elementCount - 1 DO 
		
		hr := F_VN_GetAt_TcVnVector4_DINT(TargetContainer, _value.Value, i, S_OK);
		
		IF SUCCEEDED(hr) THEN
			Serializer.AddObject(_value);
		ELSE
			Serializer.AddNull();
		END_IF
		
	END_FOR
END_IF

Serializer.EndArray();
END_METHOD

METHOD PRIVATE Serialize_ContainerType_Vector_TcVnVector4_INT
VAR_INPUT
	Serializer : I_Serializer;
	TargetContainer : ITcVnContainer;
END_VAR
VAR
	hr : HRESULT;
	_value : _TcVnVector4_INT();
	elementCount : ULINT;
	i : ULINT;
END_VAR
TargetContainer.GetElementNum(elementCount);
Serializer.StartArray();

IF elementCount > 0 THEN
	FOR i := 0 TO elementCount - 1 DO 
		
		hr := F_VN_GetAt_TcVnVector4_INT(TargetContainer, _value.Value, i, S_OK);
		
		IF SUCCEEDED(hr) THEN
			Serializer.AddObject(_value);
		ELSE
			Serializer.AddNull();
		END_IF
		
	END_FOR
END_IF

Serializer.EndArray();
END_METHOD

METHOD PRIVATE Serialize_ContainerType_Vector_TcVnVector4_LREAL
VAR_INPUT
	Serializer : I_Serializer;
	TargetContainer : ITcVnContainer;
END_VAR
VAR
	hr : HRESULT;
	_value : _TcVnVector4_LREAL();
	elementCount : ULINT;
	i : ULINT;
END_VAR
TargetContainer.GetElementNum(elementCount);
Serializer.StartArray();

IF elementCount > 0 THEN
	FOR i := 0 TO elementCount - 1 DO 
		
		hr := F_VN_GetAt_TcVnVector4_LREAL(TargetContainer, _value.Value, i, S_OK);
		
		IF SUCCEEDED(hr) THEN
			Serializer.AddObject(_value);
		ELSE
			Serializer.AddNull();
		END_IF
		
	END_FOR
END_IF

Serializer.EndArray();
END_METHOD

METHOD PRIVATE Serialize_ContainerType_Vector_TcVnVector4_REAL
VAR_INPUT
	Serializer : I_Serializer;
	TargetContainer : ITcVnContainer;
END_VAR
VAR
	hr : HRESULT;
	_value : _TcVnVector4_REAL();
	elementCount : ULINT;
	i : ULINT;
END_VAR
TargetContainer.GetElementNum(elementCount);
Serializer.StartArray();

IF elementCount > 0 THEN
	FOR i := 0 TO elementCount - 1 DO 
		
		hr := F_VN_GetAt_TcVnVector4_REAL(TargetContainer, _value.Value, i, S_OK);
		
		IF SUCCEEDED(hr) THEN
			Serializer.AddObject(_value);
		ELSE
			Serializer.AddNull();
		END_IF
		
	END_FOR
END_IF

Serializer.EndArray();
END_METHOD

METHOD PRIVATE Serialize_ContainerType_Vector_TcVnVector4_SINT
VAR_INPUT
	Serializer : I_Serializer;
	TargetContainer : ITcVnContainer;
END_VAR
VAR
	hr : HRESULT;
	_value : _TcVnVector4_SINT();
	elementCount : ULINT;
	i : ULINT;
END_VAR
TargetContainer.GetElementNum(elementCount);
Serializer.StartArray();

IF elementCount > 0 THEN
	FOR i := 0 TO elementCount - 1 DO 
		
		hr := F_VN_GetAt_TcVnVector4_SINT(TargetContainer, _value.Value, i, S_OK);
		
		IF SUCCEEDED(hr) THEN
			Serializer.AddObject(_value);
		ELSE
			Serializer.AddNull();
		END_IF
		
	END_FOR
END_IF

Serializer.EndArray();
END_METHOD

METHOD PRIVATE Serialize_ContainerType_Vector_TcVnVector4_UINT
VAR_INPUT
	Serializer : I_Serializer;
	TargetContainer : ITcVnContainer;
END_VAR
VAR
	hr : HRESULT;
	_value : _TcVnVector4_UINT();
	elementCount : ULINT;
	i : ULINT;
END_VAR
TargetContainer.GetElementNum(elementCount);
Serializer.StartArray();

IF elementCount > 0 THEN
	FOR i := 0 TO elementCount - 1 DO 
		
		hr := F_VN_GetAt_TcVnVector4_UINT(TargetContainer, _value.Value, i, S_OK);
		
		IF SUCCEEDED(hr) THEN
			Serializer.AddObject(_value);
		ELSE
			Serializer.AddNull();
		END_IF
		
	END_FOR
END_IF

Serializer.EndArray();
END_METHOD

METHOD PRIVATE Serialize_ContainerType_Vector_TcVnVector4_USINT
VAR_INPUT
	Serializer : I_Serializer;
	TargetContainer : ITcVnContainer;
END_VAR
VAR
	hr : HRESULT;
	_value : _TcVnVector4_USINT();
	elementCount : ULINT;
	i : ULINT;
END_VAR
TargetContainer.GetElementNum(elementCount);
Serializer.StartArray();

IF elementCount > 0 THEN
	FOR i := 0 TO elementCount - 1 DO 
		
		hr := F_VN_GetAt_TcVnVector4_USINT(TargetContainer, _value.Value, i, S_OK);
		
		IF SUCCEEDED(hr) THEN
			Serializer.AddObject(_value);
		ELSE
			Serializer.AddNull();
		END_IF
		
	END_FOR
END_IF

Serializer.EndArray();
END_METHOD

METHOD PRIVATE Serialize_ContainerType_Vector_UDINT
VAR_INPUT
	Serializer : I_Serializer;
	TargetContainer : ITcVnContainer;
END_VAR
VAR
	hr : HRESULT;
	_value : _UDINT(0);
	elementCount : ULINT;
	i : ULINT;
END_VAR
TargetContainer.GetElementNum(elementCount);
Serializer.StartArray();

IF elementCount > 0 THEN
	FOR i := 0 TO elementCount - 1 DO 
		
		hr := F_VN_GetAt_UDINT(TargetContainer, _value.Value, i, S_OK);
		
		IF SUCCEEDED(hr) THEN
			Serializer.AddObject(_value);
		ELSE
			Serializer.AddNull();
		END_IF
		
	END_FOR
END_IF

Serializer.EndArray();
END_METHOD

METHOD PRIVATE Serialize_ContainerType_Vector_UINT
VAR_INPUT
	Serializer : I_Serializer;
	TargetContainer : ITcVnContainer;
END_VAR
VAR
	hr : HRESULT;
	_value : _UINT(0);
	elementCount : ULINT;
	i : ULINT;
END_VAR
TargetContainer.GetElementNum(elementCount);
Serializer.StartArray();

IF elementCount > 0 THEN
	FOR i := 0 TO elementCount - 1 DO 
		
		hr := F_VN_GetAt_UINT(TargetContainer, _value.Value, i, S_OK);
		
		IF SUCCEEDED(hr) THEN
			Serializer.AddObject(_value);
		ELSE
			Serializer.AddNull();
		END_IF
		
	END_FOR
END_IF

Serializer.EndArray();
END_METHOD

METHOD PRIVATE Serialize_ContainerType_Vector_ULINT
VAR_INPUT
	Serializer : I_Serializer;
	TargetContainer : ITcVnContainer;
END_VAR
VAR
	hr : HRESULT;
	_value : _ULINT(0);
	elementCount : ULINT;
	i : ULINT;
END_VAR
TargetContainer.GetElementNum(elementCount);
Serializer.StartArray();

IF elementCount > 0 THEN
	FOR i := 0 TO elementCount - 1 DO 
		
		hr := F_VN_GetAt_ULINT(TargetContainer, _value.Value, i, S_OK);
		
		IF SUCCEEDED(hr) THEN
			Serializer.AddObject(_value);
		ELSE
			Serializer.AddNull();
		END_IF
		
	END_FOR
END_IF

Serializer.EndArray();
END_METHOD

METHOD PRIVATE Serialize_ContainerType_Vector_USINT
VAR_INPUT
	Serializer : I_Serializer;
	TargetContainer : ITcVnContainer;
END_VAR
VAR
	hr : HRESULT;
	_value : _USINT(0);
	elementCount : ULINT;
	i : ULINT;
END_VAR
TargetContainer.GetElementNum(elementCount);
Serializer.StartArray();

IF elementCount > 0 THEN
	FOR i := 0 TO elementCount - 1 DO 
		
		hr := F_VN_GetAt_USINT(TargetContainer, _value.Value, i, S_OK);
		
		IF SUCCEEDED(hr) THEN
			Serializer.AddObject(_value);
		ELSE
			Serializer.AddNull();
		END_IF
		
	END_FOR
END_IF

Serializer.EndArray();
END_METHOD

METHOD PRIVATE Serialize_ContainerType_Vector_Vector_DINT
VAR_INPUT
	Serializer : I_Serializer;
	TargetContainer : ITcVnContainer;
END_VAR
VAR
	hr : HRESULT;
	container : ITcVnContainer;
	elementCount : ULINT;
	i : ULINT;
END_VAR
TargetContainer.GetElementNum(elementCount);
Serializer.StartArray();

IF elementCount > 0 THEN
	FOR i := 0 TO elementCount - 1 DO 
		
		hr := F_VN_GetAt_ITcVnContainer(TargetContainer, container, i, S_OK);
		
		IF SUCCEEDED(hr) THEN
			Serialize_ContainerType_Vector_DINT(Serializer, container);
		ELSE
			Serializer.AddNull();
		END_IF
		
	END_FOR
END_IF

IF container <> 0 THEN
	container.TcRelease();
END_IF

Serializer.EndArray();
END_METHOD

METHOD PRIVATE Serialize_ContainerType_Vector_Vector_LREAL
VAR_INPUT
	Serializer : I_Serializer;
	TargetContainer : ITcVnContainer;
END_VAR
VAR
	hr : HRESULT;
	container : ITcVnContainer;
	elementCount : ULINT;
	i : ULINT;
END_VAR
TargetContainer.GetElementNum(elementCount);
Serializer.StartArray();

IF elementCount > 0 THEN
	FOR i := 0 TO elementCount - 1 DO 
		
		hr := F_VN_GetAt_ITcVnContainer(TargetContainer, container, i, S_OK);
		
		IF SUCCEEDED(hr) THEN
			Serialize_ContainerType_Vector_LREAL(Serializer, container);
		ELSE
			Serializer.AddNull();
		END_IF
		
	END_FOR
END_IF

IF container <> 0 THEN
	container.TcRelease();
END_IF

Serializer.EndArray();
END_METHOD

METHOD PRIVATE Serialize_ContainerType_Vector_Vector_REAL
VAR_INPUT
	Serializer : I_Serializer;
	TargetContainer : ITcVnContainer;
END_VAR
VAR
	hr : HRESULT;
	container : ITcVnContainer;
	elementCount : ULINT;
	i : ULINT;
END_VAR
TargetContainer.GetElementNum(elementCount);
Serializer.StartArray();

IF elementCount > 0 THEN
	FOR i := 0 TO elementCount - 1 DO 
		
		hr := F_VN_GetAt_ITcVnContainer(TargetContainer, container, i, S_OK);
		
		IF SUCCEEDED(hr) THEN
			Serialize_ContainerType_Vector_REAL(Serializer, container);
		ELSE
			Serializer.AddNull();
		END_IF
		
	END_FOR
END_IF

IF container <> 0 THEN
	container.TcRelease();
END_IF

Serializer.EndArray();
END_METHOD

METHOD PRIVATE Serialize_ContainerType_Vector_Vector_TcVnPoint2_DINT
VAR_INPUT
	Serializer : I_Serializer;
	TargetContainer : ITcVnContainer;
END_VAR
VAR
	hr : HRESULT;
	container : ITcVnContainer;
	elementCount : ULINT;
	i : ULINT;
END_VAR
TargetContainer.GetElementNum(elementCount);
Serializer.StartArray();

IF elementCount > 0 THEN
	FOR i := 0 TO elementCount - 1 DO 
		
		hr := F_VN_GetAt_ITcVnContainer(TargetContainer, container, i, S_OK);
		
		IF SUCCEEDED(hr) THEN
			Serialize_ContainerType_Vector_TcVnPoint2_DINT(Serializer, container);
		ELSE
			Serializer.AddNull();
		END_IF
		
	END_FOR
END_IF

IF container <> 0 THEN
	container.TcRelease();
END_IF

Serializer.EndArray();
END_METHOD

METHOD PRIVATE Serialize_ContainerType_Vector_Vector_TcVnPoint2_REAL
VAR_INPUT
	Serializer : I_Serializer;
	TargetContainer : ITcVnContainer;
END_VAR
VAR
	hr : HRESULT;
	container : ITcVnContainer;
	elementCount : ULINT;
	i : ULINT;
END_VAR
TargetContainer.GetElementNum(elementCount);
Serializer.StartArray();

IF elementCount > 0 THEN
	FOR i := 0 TO elementCount - 1 DO 
		
		hr := F_VN_GetAt_ITcVnContainer(TargetContainer, container, i, S_OK);
		
		IF SUCCEEDED(hr) THEN
			Serialize_ContainerType_Vector_TcVnPoint2_REAL(Serializer, container);
		ELSE
			Serializer.AddNull();
		END_IF
		
	END_FOR
END_IF

IF container <> 0 THEN
	container.TcRelease();
END_IF

Serializer.EndArray();
END_METHOD

METHOD PRIVATE Serialize_ContainerType_Vector_Vector_TcVnPoint3_REAL
VAR_INPUT
	Serializer : I_Serializer;
	TargetContainer : ITcVnContainer;
END_VAR
VAR
	hr : HRESULT;
	container : ITcVnContainer;
	elementCount : ULINT;
	i : ULINT;
END_VAR
TargetContainer.GetElementNum(elementCount);
Serializer.StartArray();

IF elementCount > 0 THEN
	FOR i := 0 TO elementCount - 1 DO 
		
		hr := F_VN_GetAt_ITcVnContainer(TargetContainer, container, i, S_OK);
		
		IF SUCCEEDED(hr) THEN
			Serialize_ContainerType_Vector_TcVnPoint3_REAL(Serializer, container);
		ELSE
			Serializer.AddNull();
		END_IF
		
	END_FOR
END_IF

IF container <> 0 THEN
	container.TcRelease();
END_IF

Serializer.EndArray();
END_METHOD

METHOD PRIVATE Serialize_ContainerType_Vector_Vector_UDINT
VAR_INPUT
	Serializer : I_Serializer;
	TargetContainer : ITcVnContainer;
END_VAR
VAR
	hr : HRESULT;
	container : ITcVnContainer;
	elementCount : ULINT;
	i : ULINT;
END_VAR
TargetContainer.GetElementNum(elementCount);
Serializer.StartArray();

IF elementCount > 0 THEN
	FOR i := 0 TO elementCount - 1 DO 
		
		hr := F_VN_GetAt_ITcVnContainer(TargetContainer, container, i, S_OK);
		
		IF SUCCEEDED(hr) THEN
			Serialize_ContainerType_Vector_UDINT(Serializer, container);
		ELSE
			Serializer.AddNull();
		END_IF
		
	END_FOR
END_IF

IF container <> 0 THEN
	container.TcRelease();
END_IF

Serializer.EndArray();
END_METHOD

METHOD PRIVATE Serialize_ContainerType_Vector_Vector_ULINT
VAR_INPUT
	Serializer : I_Serializer;
	TargetContainer : ITcVnContainer;
END_VAR
VAR
	hr : HRESULT;
	container : ITcVnContainer;
	elementCount : ULINT;
	i : ULINT;
END_VAR
TargetContainer.GetElementNum(elementCount);
Serializer.StartArray();

IF elementCount > 0 THEN
	FOR i := 0 TO elementCount - 1 DO 
		
		hr := F_VN_GetAt_ITcVnContainer(TargetContainer, container, i, S_OK);
		
		IF SUCCEEDED(hr) THEN
			Serialize_ContainerType_Vector_ULINT(Serializer, container);
		ELSE
			Serializer.AddNull();
		END_IF
		
	END_FOR
END_IF

IF container <> 0 THEN
	container.TcRelease();
END_IF

Serializer.EndArray();
END_METHOD

METHOD PUBLIC TryTcReleaseLocal : BOOL
VAR_INPUT
END_VAR
IF localData = 0 THEN
	RETURN;
END_IF

IF localData.TcRelease() = 0 THEN
	localData := 0;
END_IF

TryTcReleaseLocal := TRUE;
END_METHOD

METHOD PUBLIC Clone : I_Datatype
VAR
    pClone : POINTER TO _ITcVnContainer;
END_VAR
pClone := __NEW(_ITcVnContainer);
Clone := pClone^;
END_METHOD

PROPERTY PUBLIC Identifier : T_MAXSTRING
GET
Identifier := 'ITcVnContainer';
END_GET
END_PROPERTY

METHOD PUBLIC MakeReferenceTo
VAR_INPUT
	ReferenceTarget : REFERENCE TO ITcVnContainer;
END_VAR
activeData REF= ReferenceTarget;
END_METHOD

METHOD PUBLIC SerializeWith
VAR_INPUT
	Serializer : I_Serializer;
END_VAR
VAR
	containerTypeName : _STRING('');
	containerTypeGuid : _GUID;
	elementTypeGuid : _GUID;
    elementNum : _ULINT(0);
    elementSize : _ULINT(0);
END_VAR
IF NOT (activeData <> 0) THEN
	Serializer.AddNull();
	RETURN;
END_IF

activeData.GetTypeName(containerTypeName.Value,UDINT_TO_UINT(containerTypeName.Size));
activeData.GetTypeGuid(containerTypeGuid.Value);
activeData.GetElementTypeGuid(elementTypeGuid.Value);
activeData.GetElementNum(elementNum.Value);
activeData.GetElementSize(elementSize.Value);

Serializer.StartObject();
Serializer.AddKeyObject('containerTypeName', containerTypeName);
Serializer.AddKeyString('containerTypeGuid', containerTypeGuid.ToString());
Serializer.AddKeyString('elementTypeGuid', elementTypeGuid.ToString());
Serializer.AddKeyObject('elementNum', elementNum);
Serializer.AddKeyObject('elementSize', elementSize);
Serializer.AddKey('elements');
// Serializer.StartArray();

IF containerTypeName.Value = 'CTcVnContainer_Vector_SINT' THEN
	Serialize_ContainerType_Vector_SINT(Serializer, activeData);		
ELSIF containerTypeName.Value = 'CTcVnContainer_Vector_USINT' THEN
	Serialize_ContainerType_Vector_USINT(Serializer, activeData);
ELSIF containerTypeName.Value = 'CTcVnContainer_Vector_INT' THEN
	Serialize_ContainerType_Vector_INT(Serializer, activeData);
ELSIF containerTypeName.Value = 'CTcVnContainer_Vector_UINT' THEN
	Serialize_ContainerType_Vector_UINT(Serializer, activeData);
ELSIF containerTypeName.Value = 'CTcVnContainer_Vector_DINT' THEN
	Serialize_ContainerType_Vector_DINT(Serializer, activeData);
ELSIF containerTypeName.Value = 'CTcVnContainer_Vector_UDINT' THEN
	Serialize_ContainerType_Vector_UDINT(Serializer, activeData);
ELSIF containerTypeName.Value = 'CTcVnContainer_Vector_ULINT' THEN
	Serialize_ContainerType_Vector_ULINT(Serializer, activeData);
ELSIF containerTypeName.Value = 'CTcVnContainer_Vector_REAL' THEN
	Serialize_ContainerType_Vector_REAL(Serializer, activeData);
ELSIF containerTypeName.Value = 'CTcVnContainer_Vector_LREAL' THEN
	Serialize_ContainerType_Vector_LREAL(Serializer, activeData);
ELSIF containerTypeName.Value = 'CTcVnContainer_Vector_ITcVnImage' THEN
	Serialize_ContainerType_Vector_ITcVnImage(Serializer, activeData);
	
//Vector_TcVnPoint2
ELSIF containerTypeName.Value = 'CTcVnContainer_Vector_TcVnPoint2_DINT' THEN
	Serialize_ContainerType_Vector_TcVnPoint2_DINT(Serializer, activeData);
ELSIF containerTypeName.Value = 'CTcVnContainer_Vector_TcVnPoint2_REAL' THEN
	Serialize_ContainerType_Vector_TcVnPoint2_REAL(Serializer, activeData);
ELSIF containerTypeName.Value = 'CTcVnContainer_Vector_TcVnPoint2_LREAL' THEN
	Serialize_ContainerType_Vector_TcVnPoint2_LREAL(Serializer, activeData);
	
//Vector_TcVnPoint3
ELSIF containerTypeName.Value = 'CTcVnContainer_Vector_TcVnPoint3_REAL' THEN
	Serialize_ContainerType_Vector_TcVnPoint3_REAL(Serializer, activeData);
ELSIF containerTypeName.Value = 'CTcVnContainer_Vector_TcVnPoint3_LREAL' THEN
	Serialize_ContainerType_Vector_TcVnPoint3_LREAL(Serializer, activeData);
	
//Vector_TcVnVector2
ELSIF containerTypeName.Value = 'CTcVnContainer_Vector_TcVnVector2_SINT' THEN
	Serialize_ContainerType_Vector_TcVnVector2_SINT(Serializer, activeData);
ELSIF containerTypeName.Value = 'CTcVnContainer_Vector_TcVnVector2_USINT' THEN
	Serialize_ContainerType_Vector_TcVnVector2_USINT(Serializer, activeData);
ELSIF containerTypeName.Value = 'CTcVnContainer_Vector_TcVnVector2_INT' THEN
	Serialize_ContainerType_Vector_TcVnVector2_INT(Serializer, activeData);
ELSIF containerTypeName.Value = 'CTcVnContainer_Vector_TcVnVector2_UINT' THEN
	Serialize_ContainerType_Vector_TcVnVector2_UINT(Serializer, activeData);
ELSIF containerTypeName.Value = 'CTcVnContainer_Vector_TcVnVector2_DINT' THEN
	Serialize_ContainerType_Vector_TcVnVector2_DINT(Serializer, activeData);
ELSIF containerTypeName.Value = 'CTcVnContainer_Vector_TcVnVector2_REAL' THEN
	Serialize_ContainerType_Vector_TcVnVector2_REAL(Serializer, activeData);
	
//Vector_TcVnVector3
ELSIF containerTypeName.Value = 'CTcVnContainer_Vector_TcVnVector3_SINT' THEN
	Serialize_ContainerType_Vector_TcVnVector3_SINT(Serializer, activeData);
ELSIF containerTypeName.Value = 'CTcVnContainer_Vector_TcVnVector3_USINT' THEN
	Serialize_ContainerType_Vector_TcVnVector3_USINT(Serializer, activeData);
ELSIF containerTypeName.Value = 'CTcVnContainer_Vector_TcVnVector3_INT' THEN
	Serialize_ContainerType_Vector_TcVnVector3_INT(Serializer, activeData);
ELSIF containerTypeName.Value = 'CTcVnContainer_Vector_TcVnVector3_UINT' THEN
	Serialize_ContainerType_Vector_TcVnVector3_UINT(Serializer, activeData);
ELSIF containerTypeName.Value = 'CTcVnContainer_Vector_TcVnVector3_REAL' THEN
	Serialize_ContainerType_Vector_TcVnVector3_REAL(Serializer, activeData);
	
//Vector_TcVnVector4
ELSIF containerTypeName.Value = 'CTcVnContainer_Vector_TcVnVector4_SINT' THEN
	Serialize_ContainerType_Vector_TcVnVector4_SINT(Serializer, activeData);
ELSIF containerTypeName.Value = 'CTcVnContainer_Vector_TcVnVector4_USINT' THEN
	Serialize_ContainerType_Vector_TcVnVector4_USINT(Serializer, activeData);
ELSIF containerTypeName.Value = 'CTcVnContainer_Vector_TcVnVector4_INT' THEN
	Serialize_ContainerType_Vector_TcVnVector4_INT(Serializer, activeData);
ELSIF containerTypeName.Value = 'CTcVnContainer_Vector_TcVnVector4_UINT' THEN
	Serialize_ContainerType_Vector_TcVnVector4_UINT(Serializer, activeData);
ELSIF containerTypeName.Value = 'CTcVnContainer_Vector_TcVnVector4_DINT' THEN
	Serialize_ContainerType_Vector_TcVnVector4_DINT(Serializer, activeData);
ELSIF containerTypeName.Value = 'CTcVnContainer_Vector_TcVnVector4_REAL' THEN
	Serialize_ContainerType_Vector_TcVnVector4_REAL(Serializer, activeData);
ELSIF containerTypeName.Value = 'CTcVnContainer_Vector_TcVnVector4_LREAL' THEN
	Serialize_ContainerType_Vector_TcVnVector4_LREAL(Serializer, activeData);
	
//Vector_Vector
ELSIF containerTypeName.Value = 'CTcVnContainer_Vector_Vector_DINT' THEN
	Serialize_ContainerType_Vector_Vector_DINT(Serializer, activeData);
ELSIF containerTypeName.Value = 'CTcVnContainer_Vector_Vector_UDINT' THEN
	Serialize_ContainerType_Vector_Vector_UDINT(Serializer, activeData);
ELSIF containerTypeName.Value = 'CTcVnContainer_Vector_Vector_ULINT' THEN
	Serialize_ContainerType_Vector_Vector_ULINT(Serializer, activeData);
ELSIF containerTypeName.Value = 'CTcVnContainer_Vector_Vector_REAL' THEN
	Serialize_ContainerType_Vector_Vector_REAL(Serializer, activeData);
ELSIF containerTypeName.Value = 'CTcVnContainer_Vector_Vector_LREAL' THEN
	Serialize_ContainerType_Vector_Vector_LREAL(Serializer, activeData);
	
//Vector_Vector_TcVnPoint2
ELSIF containerTypeName.Value = 'CTcVnContainer_Vector_Vector_TcVnPoint2_DINT' THEN
	Serialize_ContainerType_Vector_Vector_TcVnPoint2_DINT(Serializer, activeData);	
ELSIF containerTypeName.Value = 'CTcVnContainer_Vector_Vector_TcVnPoint2_REAL' THEN
	Serialize_ContainerType_Vector_Vector_TcVnPoint2_REAL(Serializer, activeData);
	
//Vector_Vector_TcVnPoint3	
ELSIF containerTypeName.Value = 'CTcVnContainer_Vector_Vector_TcVnPoint3_REAL' THEN
	Serialize_ContainerType_Vector_Vector_TcVnPoint3_REAL(Serializer, activeData);
	
//Other
ELSIF containerTypeName.Value = 'CTcVnContainer_Vector_TcVnRectangle_DINT' THEN
	Serialize_ContainerType_Vector_TcVnRectangle_DINT(Serializer, activeData);
ELSIF containerTypeName.Value = 'CTcVnContainer_Vector_TcVnRotatedRectangle' THEN
	Serialize_ContainerType_Vector_TcVnRotatedRectangle(Serializer, activeData);
ELSIF containerTypeName.Value = 'CTcVnContainer_Vector_TcVnKeyPoint' THEN
	Serialize_ContainerType_Vector_TcVnKeyPoint(Serializer, activeData);
ELSIF containerTypeName.Value = 'CTcVnContainer_Vector_TcVnDMatch' THEN
	Serialize_ContainerType_Vector_TcVnDMatch(Serializer, activeData);
ELSIF containerTypeName.Value = 'CTcVnContainer_Vector_Vector_TcVnDMatch' THEN
	Serialize_ContainerType_Vector_TcVnDMatch(Serializer, activeData);
ELSIF containerTypeName.Value = 'CTcVnContainer_String_SINT' THEN
	Serialize_ContainerType_String_SINT(Serializer, activeData);
ELSIF containerTypeName.Value = 'CTcVnContainer_Vector_String_SINT' THEN
	Serialize_ContainerType_Vector_String_SINT(Serializer, activeData);
		
END_IF
// Serializer.EndArray();
Serializer.EndObject();
END_METHOD

METHOD TryDeserializeFrom : BOOL
VAR_INPUT
	Deserializer : I_Deserializer;
	Feedback : I_DeserializerFeedback;
END_VAR
VAR
END_VAR
// not yet implemented.  This will just be a reverse of the serialization code.
END_METHOD

METHOD TryMakeReferenceTo : BOOL
VAR_INPUT
	Target : I_Datatype;
END_VAR
VAR
	pTargetData : POINTER TO ITcVnContainer;
END_VAR
IF NOT IsEquivalentTo(Target) THEN
	RETURN;
END_IF

pTargetData := Target.Address;
activeData REF= pTargetData^;
TryMakeReferenceTo := TRUE;
END_METHOD

PROPERTY PUBLIC Value : REFERENCE TO ITcVnContainer
GET
Value REF= activeData;
END_GET
END_PROPERTY

METHOD PUBLIC IsType : BOOL
VAR_INPUT
	ContainerType : GUID;
END_VAR
VAR
    actualGuid : GUID;
END_VAR
IF NOT IsValid THEN
    RETURN;
END_IF

IF NOT SUCCEEDED(activeData.GetTypeGuid(actualGuid)) THEN
    RETURN;
END_IF

IF NOT (GuidsEqualByVal(ContainerType, actualGuid)) THEN
	RETURN;
END_IF

IsType := TRUE;
END_METHOD

PROPERTY PUBLIC IsValid : BOOL
GET
IsValid := activeData <> 0;
END_GET
END_PROPERTY

METHOD PUBLIC TryCheckIfBasicContainer : BOOL
VAR_INPUT
	Result : REFERENCE TO BOOL;
END_VAR
Result := FALSE;

IF NOT IsValid THEN
	RETURN;
END_IF

IF activeData.CheckIfBasicContainer() = S_OK THEN
    Result := TRUE;
END_IF

TryCheckIfBasicContainer := TRUE;
END_METHOD

METHOD PUBLIC TryCheckIfEmpty : BOOL
VAR_INPUT
	Result : REFERENCE TO BOOL;
END_VAR
Result := FALSE;

IF NOT IsValid THEN
	RETURN;
END_IF

IF activeData.CheckIfEmpty() = S_OK THEN
    Result := TRUE;
END_IF

TryCheckIfEmpty := TRUE;
END_METHOD

METHOD PUBLIC TryCopyContentFrom : BOOL
VAR_INPUT
	Source : I_InterfaceDatatype;
END_VAR
VAR
	ipSrcContainer : I_InterfaceDatatype_ITcVnContainer;
	hresult : HRESULT;
END_VAR
IF NOT __QUERYINTERFACE(Source, ipSrcContainer) THEN
	RETURN;
END_IF

hresult := F_VN_CopyContainer(
    ipSrcContainer := ipSrcContainer.Value,
	ipDestContainer := Value,
	hrPrev:= S_OK);
    
TryCopyContentFrom := SUCCEEDED(hresult);
END_METHOD

METHOD PUBLIC TryGetElementNum : BOOL
VAR_INPUT
	Destination : REFERENCE TO ULINT;
END_VAR
IF NOT IsValid THEN
	RETURN;
END_IF

TryGetElementNum := SUCCEEDED(activeData.GetElementNum(Destination));
END_METHOD

METHOD PUBLIC TryGetElementSize : BOOL
VAR_INPUT
	Destination : REFERENCE TO ULINT;
END_VAR
IF NOT IsValid THEN
	RETURN;
END_IF

TryGetElementSize := SUCCEEDED(activeData.GetElementSize(Destination));
END_METHOD

METHOD PUBLIC TryGetElementTypeGuid : BOOL
VAR_INPUT
	Destination : REFERENCE TO GUID;
END_VAR
IF NOT IsValid THEN
	RETURN;
END_IF

TryGetElementTypeGuid := SUCCEEDED(activeData.GetElementTypeGuid(Destination));
END_METHOD

METHOD PUBLIC TryGetExportSize : BOOL
VAR_INPUT
	Destination : REFERENCE TO ULINT;
END_VAR
IF NOT IsValid THEN
	RETURN;
END_IF

TryGetExportSize := SUCCEEDED(activeData.GetExportSize(Destination));
END_METHOD

METHOD PUBLIC TryGetTypeName : BOOL
VAR_INPUT
	Destination : REFERENCE TO STRING;
END_VAR
IF NOT IsValid THEN
	RETURN;
END_IF

TryGetTypeName := SUCCEEDED(activeData.GetTypeName(Destination, 255));
END_METHOD

METHOD PUBLIC TryTcAddRef : BOOL
VAR_INPUT
END_VAR
IF activeData = 0 THEN
	RETURN;
END_IF

IF activeData.TcAddRef() = 0 THEN
	activeData := 0;
END_IF

TryTcAddRef := TRUE;
END_METHOD

METHOD PUBLIC TryTcRelease : BOOL
VAR_INPUT
END_VAR
IF activeData = 0 THEN
	RETURN;
END_IF

IF activeData.TcRelease() = 0 THEN
	activeData := 0;
END_IF

TryTcRelease := TRUE;
END_METHOD

END_FUNCTION_BLOCK

// Datatypes/Interfaces/Containers/ITcVnContainer/I_InterfaceDatatype_ITcVnContainer
INTERFACE I_InterfaceDatatype_ITcVnContainer EXTENDS I_InterfaceDatatype

PROPERTY PUBLIC Value : REFERENCE TO ITcVnContainer
GET
END_GET
END_PROPERTY

END_INTERFACE

// Datatypes/Structs/_TcVnDMatch
{attribute 'linkalways'} 
{attribute 'no_explicit_call' := 'This FB is a CLASS and must be accessed using methods or properties'}
{attribute 'enable_dynamic_creation'}
FUNCTION_BLOCK _TcVnDMatch EXTENDS StructuredDatatypeBase
VAR
	localData : TcVnDMatch;
	activeData : REFERENCE TO TcVnDMatch REF= localData;
    _nQueryIdx : _DINT(localdata.nQueryIdx);
    _nTrainIdx : _DINT(localdata.nTrainIdx);
    _nImageIdx : _DINT(localdata.nImageIdx);
    _fDistance : _REAL(localdata.fDistance);
END_VAR

PROPERTY PUBLIC Address : PVOID
GET
Address := ADR(activeData);
END_GET
END_PROPERTY

METHOD PUBLIC ClearReference
VAR_INPUT
END_VAR
activeData REF= localData;
SetMemberReference();
END_METHOD

PROPERTY PUBLIC Size : UDINT
GET
Size := SIZEOF(activeData);
END_GET
END_PROPERTY

METHOD FB_init : BOOL
VAR_INPUT
	bInitRetains : BOOL; // if TRUE, the retain variables are initialized (warm start / cold start)
	bInCopyCode : BOOL;  // if TRUE, the instance afterwards gets moved into the copy code (online change)
END_VAR
SetMemberReference();
AddMember('nQueryIdx', _nQueryIdx);
AddMember('nTrainIdx', _nTrainIdx);
AddMember('nImageIdx', _nImageIdx);
AddMember('fDistance', _fDistance);
END_METHOD

METHOD PROTECTED SetMemberReference
VAR_INPUT
END_VAR
_nQueryIdx.MakeReferenceTo(activeData.nQueryIdx);
_nTrainIdx.MakeReferenceTo(activeData.nTrainIdx);
_nImageIdx.MakeReferenceTo(activeData.nImageIdx);
_fDistance.MakeReferenceTo(activeData.fDistance);
END_METHOD

METHOD PUBLIC Clone : I_Datatype
VAR
    pClone : POINTER TO _TcVnDMatch;
END_VAR
pClone := __NEW(_TcVnDMatch());
pClone^.Value := Value;
Clone := pClone^;
END_METHOD

PROPERTY PUBLIC Identifier : T_MAXSTRING
GET
Identifier := 'TcVnDMatch';
END_GET
END_PROPERTY

METHOD PUBLIC MakeReferenceTo
VAR_INPUT
	ReferenceTarget : REFERENCE TO TcVnDMatch;
END_VAR
activeData REF= ReferenceTarget;
SetMemberReference();
END_METHOD

METHOD TryMakeReferenceTo : BOOL
VAR_INPUT
	Target : I_Datatype;
END_VAR
VAR
	targetAsStruct : I_StructuredDatatype;
	pTargetData : POINTER TO TcVnDMatch;
END_VAR
IF NOT Target.TryResolveAsStructuredDatatype(targetAsStruct) THEN
	RETURN;
END_IF

IF NOT (targetAsStruct.Identifier = Identifier) THEN
	RETURN;
END_IF

pTargetData := Target.Address;
activeData REF= pTargetData^;
SetMemberReference();
TryMakeReferenceTo := TRUE;
END_METHOD

PROPERTY PUBLIC Value : REFERENCE TO TcVnDMatch
GET
Value REF= activeData;
END_GET
END_PROPERTY

PROPERTY PUBLIC fDistance : REFERENCE TO _REAL
GET
fDistance REF= _fDistance;
END_GET
END_PROPERTY

PROPERTY PUBLIC nImageIdx : REFERENCE TO _DINT
GET
nImageIdx REF= _nImageIdx;
END_GET
END_PROPERTY

PROPERTY PUBLIC nQueryIdx : REFERENCE TO _DINT
GET
nQueryIdx REF= _nQueryIdx;
END_GET
END_PROPERTY

PROPERTY PUBLIC nTrainIdx : REFERENCE TO _DINT
GET
nTrainIdx REF= _nTrainIdx;
END_GET
END_PROPERTY

END_FUNCTION_BLOCK

